REGION Network 17: Lift01 Y-Heber / Lift01 Y-Lift
   #sinstLift01_Y_Lift(iniHomePos := "FG_TS_Lift01_Y_Lift_InHome",   // "Cylinder_2Out2In"
                       iniWorkPos := "FG_TS_Lift01_Y_Lift_InWork",
                       actor := "TransportActors".Lift01_Lift,
                       signals := #signals,
                       manualMovement := #manualMovements,
                       homePos => "FG_TS_Lift01_Y_Lift_HomePos",
                       workPos => "FG_TS_Lift01_Y_Lift_WorkPos");
END_REGION

REGION Network 18: Lift01 M-Förderband / Lift01 M-Conveyor
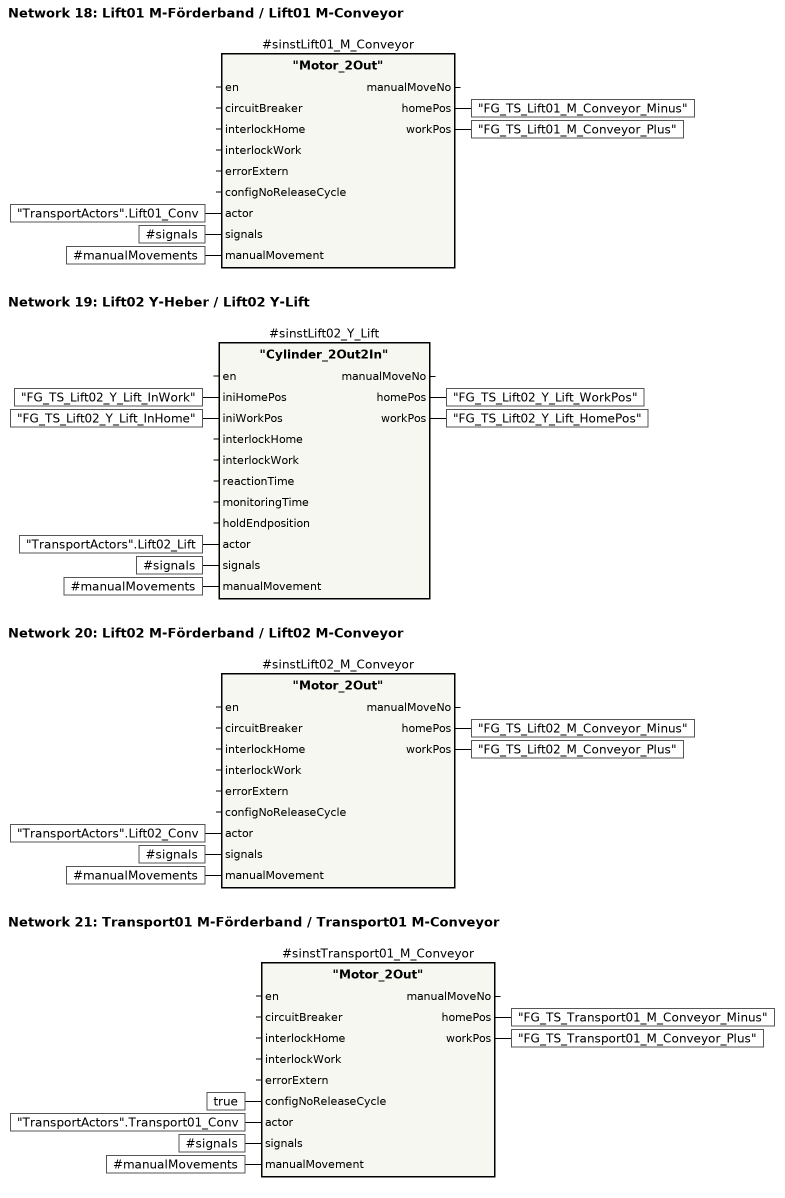
   #sinstLift01_M_Conveyor(actor := "TransportActors".Lift01_Conv,   // "Motor_2Out"
                           signals := #signals,
                           manualMovement := #manualMovements,
                           homePos => "FG_TS_Lift01_M_Conveyor_Minus",
                           workPos => "FG_TS_Lift01_M_Conveyor_Plus");
END_REGION

REGION Network 19: Lift02 Y-Heber / Lift02 Y-Lift
   #sinstLift02_Y_Lift(iniHomePos := "FG_TS_Lift02_Y_Lift_InWork",   // "Cylinder_2Out2In"
                       iniWorkPos := "FG_TS_Lift02_Y_Lift_InHome",
                       actor := "TransportActors".Lift02_Lift,
                       signals := #signals,
                       manualMovement := #manualMovements,
                       homePos => "FG_TS_Lift02_Y_Lift_WorkPos",
                       workPos => "FG_TS_Lift02_Y_Lift_HomePos");
END_REGION

REGION Network 20: Lift02 M-Förderband / Lift02 M-Conveyor
   #sinstLift02_M_Conveyor(actor := "TransportActors".Lift02_Conv,   // "Motor_2Out"
                           signals := #signals,
                           manualMovement := #manualMovements,
                           homePos => "FG_TS_Lift02_M_Conveyor_Minus",
                           workPos => "FG_TS_Lift02_M_Conveyor_Plus");
END_REGION

REGION Network 21: Transport01 M-Förderband / Transport01 M-Conveyor
   #sinstTransport01_M_Conveyor(configNoReleaseCycle := true,   // "Motor_2Out"
                           actor := "TransportActors".Transport01_Conv,
                           signals := #signals,
                           manualMovement := #manualMovements,
                           homePos => "FG_TS_Transport01_M_Conveyor_Minus",
                           workPos => "FG_TS_Transport01_M_Conveyor_Plus");
END_REGION

REGION Network 22: Transport02 M-Förderband / Transport02 M-Conveyor
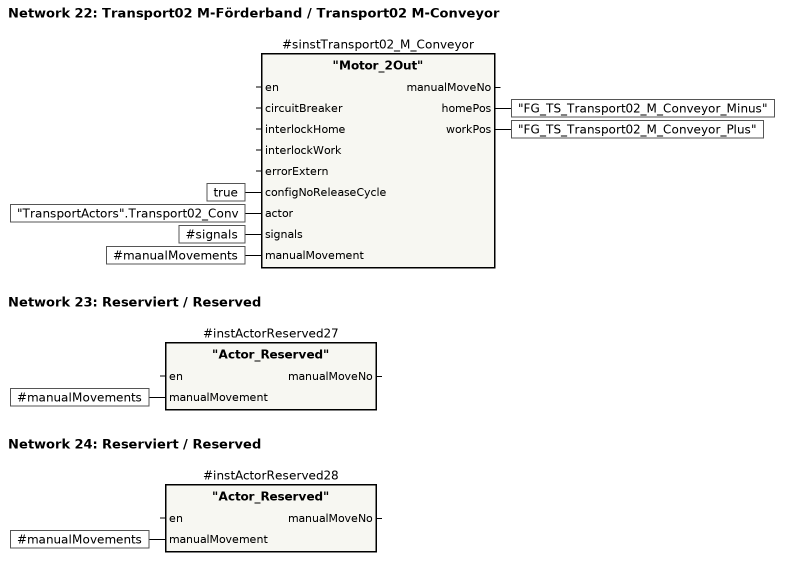
   #sinstTransport02_M_Conveyor(configNoReleaseCycle := true,   // "Motor_2Out"
                           actor := "TransportActors".Transport02_Conv,
                           signals := #signals,
                           manualMovement := #manualMovements,
                           homePos => "FG_TS_Transport02_M_Conveyor_Minus",
                           workPos => "FG_TS_Transport02_M_Conveyor_Plus");
END_REGION

REGION Network 23: Reserviert / Reserved
   #instActorReserved27(manualMovement := #manualMovements);   // "Actor_Reserved"
END_REGION

REGION Network 24: Reserviert / Reserved
   #instActorReserved28(manualMovement := #manualMovements);   // "Actor_Reserved"
END_REGION
END_FUNCTION_BLOCK

// folder: 2. Machine/10_FG_Transport/Stepsequences

FUNCTION "FG10StepSequences" : Void   // FC2010, FBD
TITLE = Schrittkettensteuerung / Sequence control
{ S7_Optimized_Access := 'TRUE' }
VERSION : 0.1
// Ersteller: Andreas Fast Automation
// Kontakt per LinkedIn: https://www.linkedin.com/in/automation-fast-andreas/
// 
// Das Projekt dient zu Demonstrationszwecken und kann frei genutzt werden.
// 
// Bausteinbeschreibung:
// Author: Andreas Fast Automation
// Kontakt per LinkedIn: https://www.linkedin.com/in/automation-fast-andreas/
// 
// This project is intended for demonstration purposes and may be used freely.
// 
// Block description:
   VAR_IN_OUT
      station : "typeStation";
   END_VAR
   VAR_TEMP
      tempInit : Bool;
      tempAck : Bool;
      tempSwAuto : Bool;
      tempSwMan : Bool;
      tempSwTap : Bool;
      tempPush : Bool;
   END_VAR
BEGIN

REGION Network 1: GRAPH-Parameter / GRAPH parameters
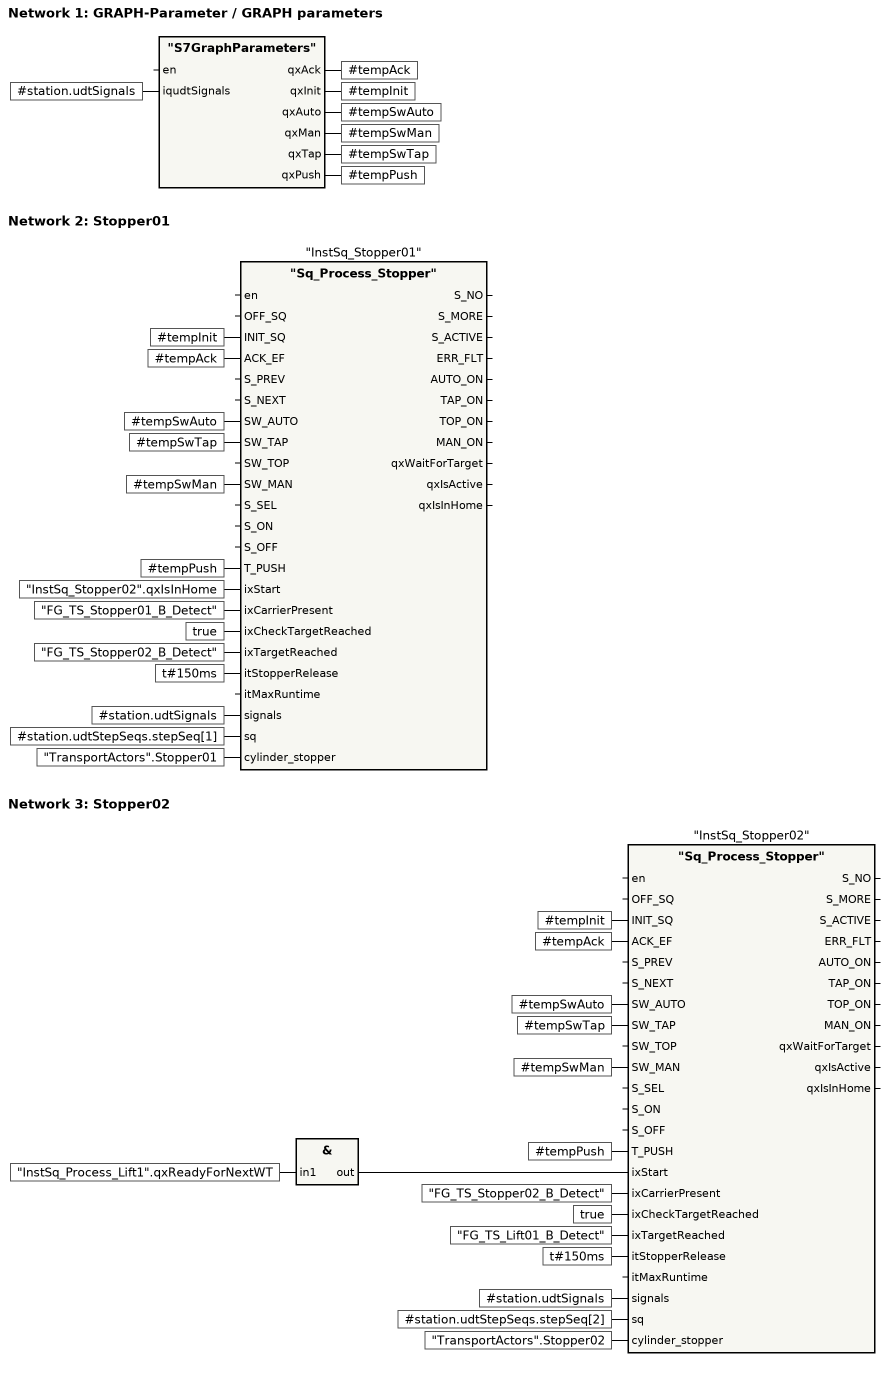
   "S7GraphParameters"(iqudtSignals := #station.udtSignals,
                       qxAck => #tempAck,
                       qxInit => #tempInit,
                       qxAuto => #tempSwAuto,
                       qxMan => #tempSwMan,
                       qxTap => #tempSwTap,
                       qxPush => #tempPush);
END_REGION

REGION Network 2: Stopper01
   "InstSq_Stopper01"(INIT_SQ := #tempInit,   // "Sq_Process_Stopper"
                      ACK_EF := #tempAck,
                      SW_AUTO := #tempSwAuto,
                      SW_TAP := #tempSwTap,
                      SW_MAN := #tempSwMan,
                      T_PUSH := #tempPush,
                      ixStart := "InstSq_Stopper02".qxIsInHome,
                      ixCarrierPresent := "FG_TS_Stopper01_B_Detect",
                      ixCheckTargetReached := true,
                      ixTargetReached := "FG_TS_Stopper02_B_Detect",
                      itStopperRelease := t#150ms,
                      signals := #station.udtSignals,
                      sq := #station.udtStepSeqs.stepSeq[1],
                      cylinder_stopper := "TransportActors".Stopper01);
END_REGION

REGION Network 3: Stopper02
   "InstSq_Stopper02"(INIT_SQ := #tempInit,   // "Sq_Process_Stopper"
                      ACK_EF := #tempAck,
                      SW_AUTO := #tempSwAuto,
                      SW_TAP := #tempSwTap,
                      SW_MAN := #tempSwMan,
                      T_PUSH := #tempPush,
                      ixStart := "InstSq_Process_Lift1".qxReadyForNextWT,
                      ixCarrierPresent := "FG_TS_Stopper02_B_Detect",
                      ixCheckTargetReached := true,
                      ixTargetReached := "FG_TS_Lift01_B_Detect",
                      itStopperRelease := t#150ms,
                      signals := #station.udtSignals,
                      sq := #station.udtStepSeqs.stepSeq[2],
                      cylinder_stopper := "TransportActors".Stopper02);
END_REGION

REGION Network 4: Lift 1
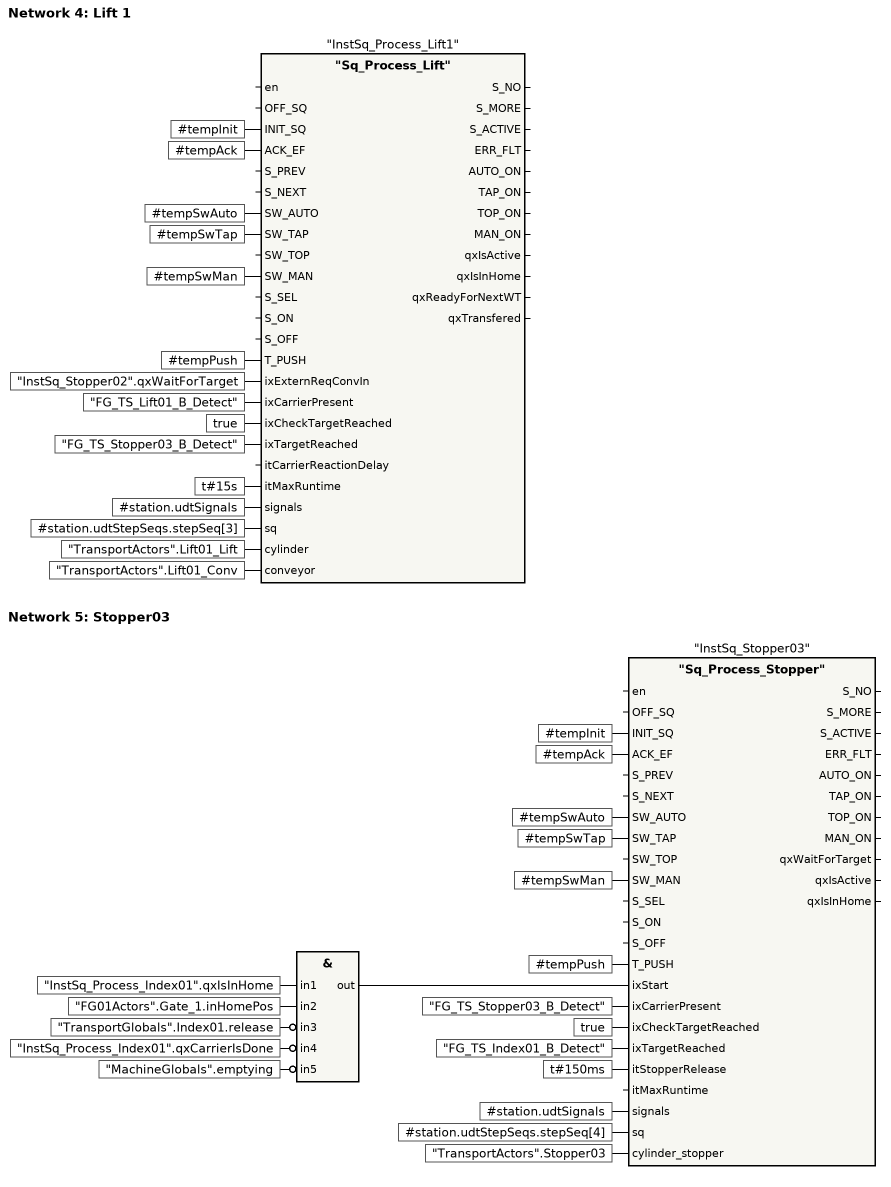
   "InstSq_Process_Lift1"(INIT_SQ := #tempInit,   // "Sq_Process_Lift"
                          ACK_EF := #tempAck,
                          SW_AUTO := #tempSwAuto,
                          SW_TAP := #tempSwTap,
                          SW_MAN := #tempSwMan,
                          T_PUSH := #tempPush,
                          ixExternReqConvIn := "InstSq_Stopper02".qxWaitForTarget,
                          ixCarrierPresent := "FG_TS_Lift01_B_Detect",
                          ixCheckTargetReached := true,
                          ixTargetReached := "FG_TS_Stopper03_B_Detect",
                          itMaxRuntime := t#15s,
                          signals := #station.udtSignals,
                          sq := #station.udtStepSeqs.stepSeq[3],
                          cylinder := "TransportActors".Lift01_Lift,
                          conveyor := "TransportActors".Lift01_Conv);
END_REGION

REGION Network 5: Stopper03
   "InstSq_Stopper03"(INIT_SQ := #tempInit,   // "Sq_Process_Stopper"
                      ACK_EF := #tempAck,
                      SW_AUTO := #tempSwAuto,
                      SW_TAP := #tempSwTap,
                      SW_MAN := #tempSwMan,
                      T_PUSH := #tempPush,
                      ixStart := "InstSq_Process_Index01".qxIsInHome AND "FG01Actors".Gate_1.inHomePos AND NOT "TransportGlobals".Index01.release AND NOT "InstSq_Process_Index01".qxCarrierIsDone AND NOT "MachineGlobals".emptying,
                      ixCarrierPresent := "FG_TS_Stopper03_B_Detect",
                      ixCheckTargetReached := true,
                      ixTargetReached := "FG_TS_Index01_B_Detect",
                      itStopperRelease := t#150ms,
                      signals := #station.udtSignals,
                      sq := #station.udtStepSeqs.stepSeq[4],
                      cylinder_stopper := "TransportActors".Stopper03);
END_REGION

REGION Network 6: Index01
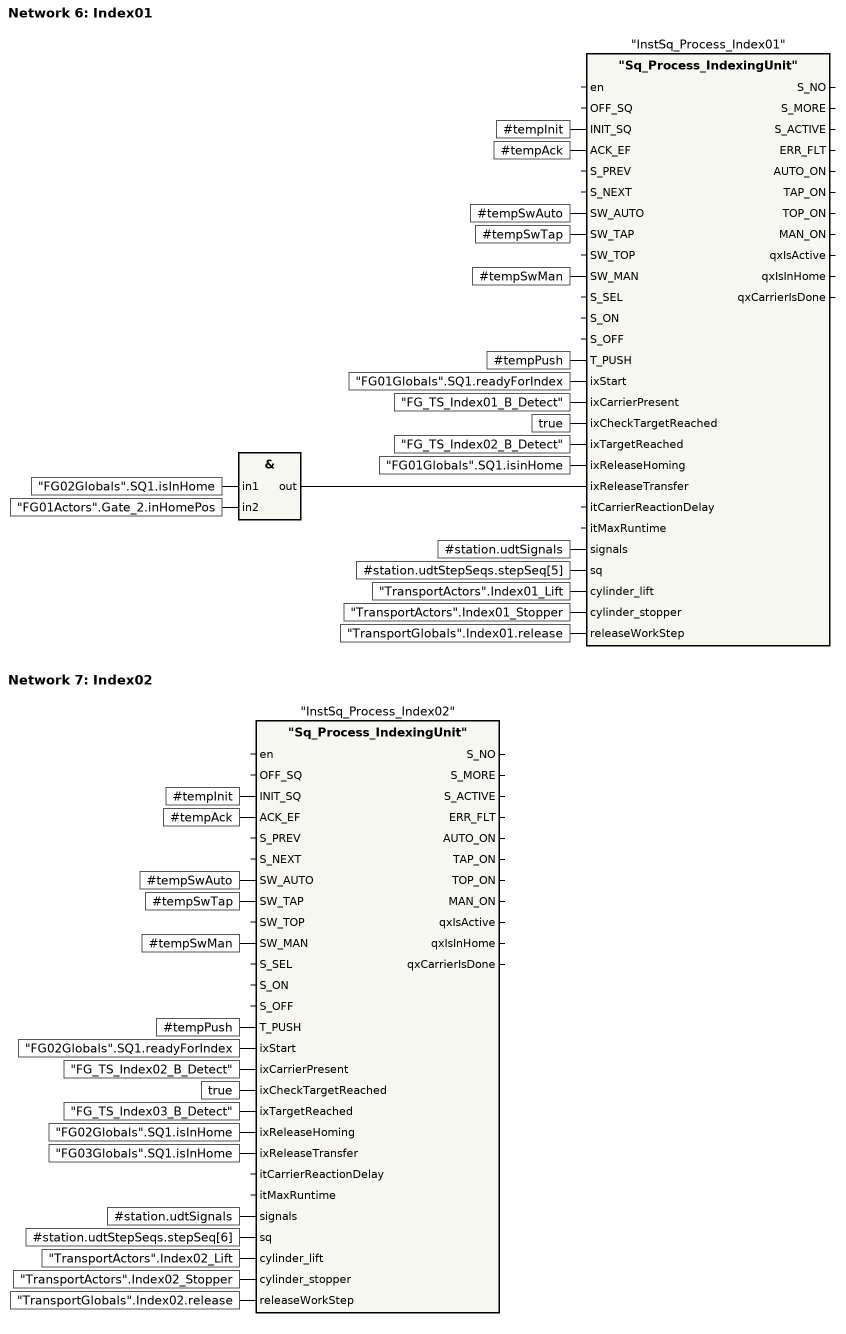
   "InstSq_Process_Index01"(INIT_SQ := #tempInit,   // "Sq_Process_IndexingUnit"
                           ACK_EF := #tempAck,
                           SW_AUTO := #tempSwAuto,
                           SW_TAP := #tempSwTap,
                           SW_MAN := #tempSwMan,
                           T_PUSH := #tempPush,
                           ixStart := "FG01Globals".SQ1.readyForIndex,
                           ixCarrierPresent := "FG_TS_Index01_B_Detect",
                           ixCheckTargetReached := true,
                           ixTargetReached := "FG_TS_Index02_B_Detect",
                           ixReleaseHoming := "FG01Globals".SQ1.isinHome,
                           ixReleaseTransfer := "FG02Globals".SQ1.isInHome AND "FG01Actors".Gate_2.inHomePos,
                           signals := #station.udtSignals,
                           sq := #station.udtStepSeqs.stepSeq[5],
                           cylinder_lift := "TransportActors".Index01_Lift,
                           cylinder_stopper := "TransportActors".Index01_Stopper,
                           releaseWorkStep := "TransportGlobals".Index01.release);
END_REGION

REGION Network 7: Index02
   "InstSq_Process_Index02"(INIT_SQ := #tempInit,   // "Sq_Process_IndexingUnit"
                           ACK_EF := #tempAck,
                           SW_AUTO := #tempSwAuto,
                           SW_TAP := #tempSwTap,
                           SW_MAN := #tempSwMan,
                           T_PUSH := #tempPush,
                           ixStart := "FG02Globals".SQ1.readyForIndex,
                           ixCarrierPresent := "FG_TS_Index02_B_Detect",
                           ixCheckTargetReached := true,
                           ixTargetReached := "FG_TS_Index03_B_Detect",
                           ixReleaseHoming := "FG02Globals".SQ1.isInHome,
                           ixReleaseTransfer := "FG03Globals".SQ1.isInHome,
                           signals := #station.udtSignals,
                           sq := #station.udtStepSeqs.stepSeq[6],
                           cylinder_lift := "TransportActors".Index02_Lift,
                           cylinder_stopper := "TransportActors".Index02_Stopper,
                           releaseWorkStep := "TransportGlobals".Index02.release);
END_REGION

REGION Network 8: Index03
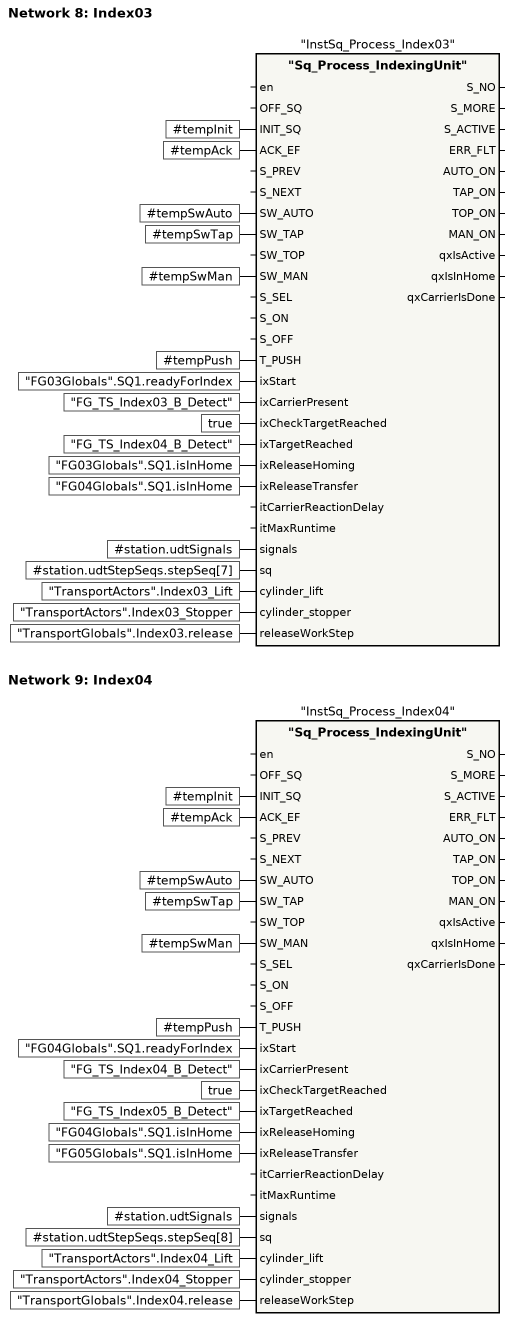
   "InstSq_Process_Index03"(INIT_SQ := #tempInit,   // "Sq_Process_IndexingUnit"
                           ACK_EF := #tempAck,
                           SW_AUTO := #tempSwAuto,
                           SW_TAP := #tempSwTap,
                           SW_MAN := #tempSwMan,
                           T_PUSH := #tempPush,
                           ixStart := "FG03Globals".SQ1.readyForIndex,
                           ixCarrierPresent := "FG_TS_Index03_B_Detect",
                           ixCheckTargetReached := true,
                           ixTargetReached := "FG_TS_Index04_B_Detect",
                           ixReleaseHoming := "FG03Globals".SQ1.isInHome,
                           ixReleaseTransfer := "FG04Globals".SQ1.isInHome,
                           signals := #station.udtSignals,
                           sq := #station.udtStepSeqs.stepSeq[7],
                           cylinder_lift := "TransportActors".Index03_Lift,
                           cylinder_stopper := "TransportActors".Index03_Stopper,
                           releaseWorkStep := "TransportGlobals".Index03.release);
END_REGION

REGION Network 9: Index04
   "InstSq_Process_Index04"(INIT_SQ := #tempInit,   // "Sq_Process_IndexingUnit"
                           ACK_EF := #tempAck,
                           SW_AUTO := #tempSwAuto,
                           SW_TAP := #tempSwTap,
                           SW_MAN := #tempSwMan,
                           T_PUSH := #tempPush,
                           ixStart := "FG04Globals".SQ1.readyForIndex,
                           ixCarrierPresent := "FG_TS_Index04_B_Detect",
                           ixCheckTargetReached := true,
                           ixTargetReached := "FG_TS_Index05_B_Detect",
                           ixReleaseHoming := "FG04Globals".SQ1.isInHome,
                           ixReleaseTransfer := "FG05Globals".SQ1.isInHome,
                           signals := #station.udtSignals,
                           sq := #station.udtStepSeqs.stepSeq[8],
                           cylinder_lift := "TransportActors".Index04_Lift,
                           cylinder_stopper := "TransportActors".Index04_Stopper,
                           releaseWorkStep := "TransportGlobals".Index04.release);
END_REGION

REGION Network 10: Index05
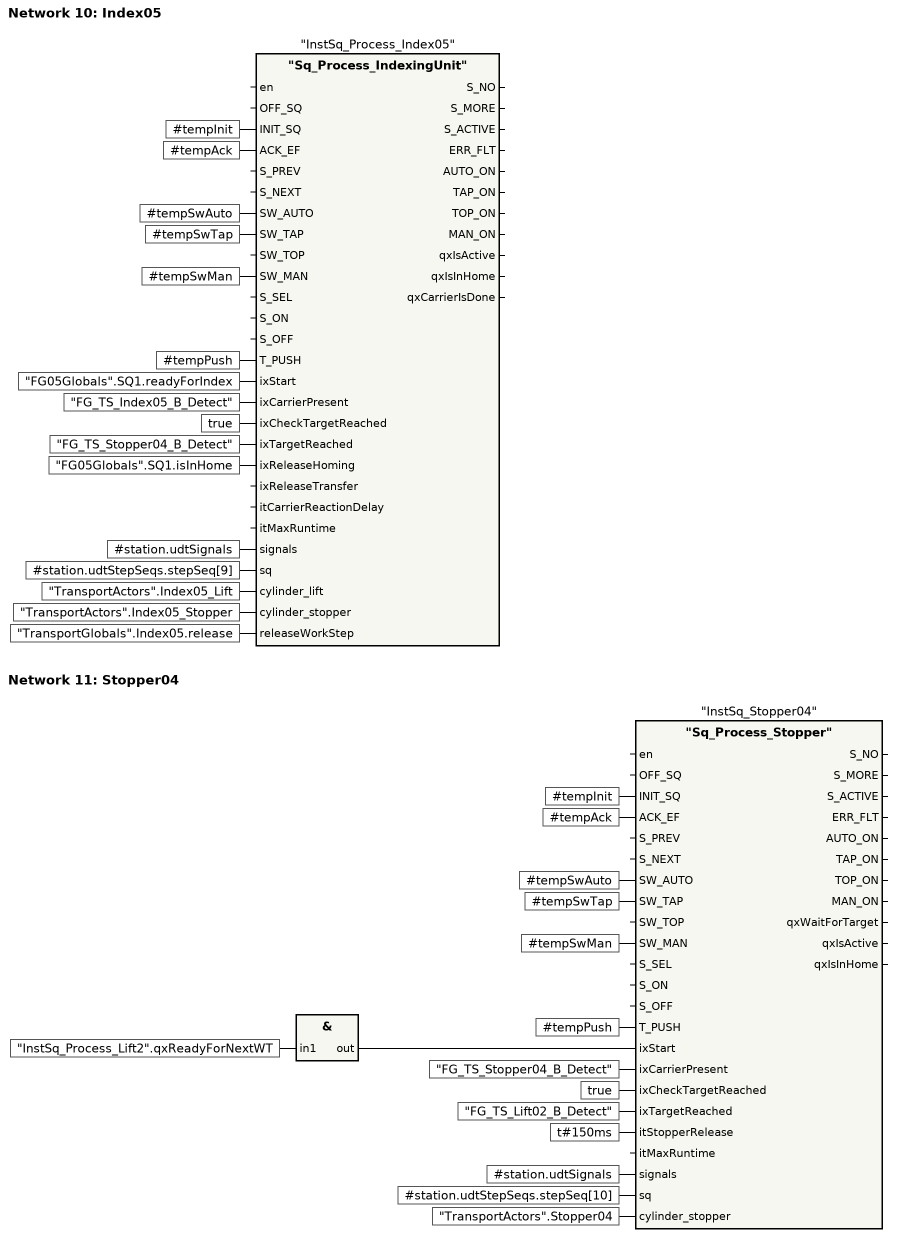
   "InstSq_Process_Index05"(INIT_SQ := #tempInit,   // "Sq_Process_IndexingUnit"
                           ACK_EF := #tempAck,
                           SW_AUTO := #tempSwAuto,
                           SW_TAP := #tempSwTap,
                           SW_MAN := #tempSwMan,
                           T_PUSH := #tempPush,
                           ixStart := "FG05Globals".SQ1.readyForIndex,
                           ixCarrierPresent := "FG_TS_Index05_B_Detect",
                           ixCheckTargetReached := true,
                           ixTargetReached := "FG_TS_Stopper04_B_Detect",
                           ixReleaseHoming := "FG05Globals".SQ1.isInHome,
                           signals := #station.udtSignals,
                           sq := #station.udtStepSeqs.stepSeq[9],
                           cylinder_lift := "TransportActors".Index05_Lift,
                           cylinder_stopper := "TransportActors".Index05_Stopper,
                           releaseWorkStep := "TransportGlobals".Index05.release);
END_REGION

REGION Network 11: Stopper04
   "InstSq_Stopper04"(INIT_SQ := #tempInit,   // "Sq_Process_Stopper"
                      ACK_EF := #tempAck,
                      SW_AUTO := #tempSwAuto,
                      SW_TAP := #tempSwTap,
                      SW_MAN := #tempSwMan,
                      T_PUSH := #tempPush,
                      ixStart := "InstSq_Process_Lift2".qxReadyForNextWT,
                      ixCarrierPresent := "FG_TS_Stopper04_B_Detect",
                      ixCheckTargetReached := true,
                      ixTargetReached := "FG_TS_Lift02_B_Detect",
                      itStopperRelease := t#150ms,
                      signals := #station.udtSignals,
                      sq := #station.udtStepSeqs.stepSeq[10],
                      cylinder_stopper := "TransportActors".Stopper04);
END_REGION

REGION Network 12: Lift 2
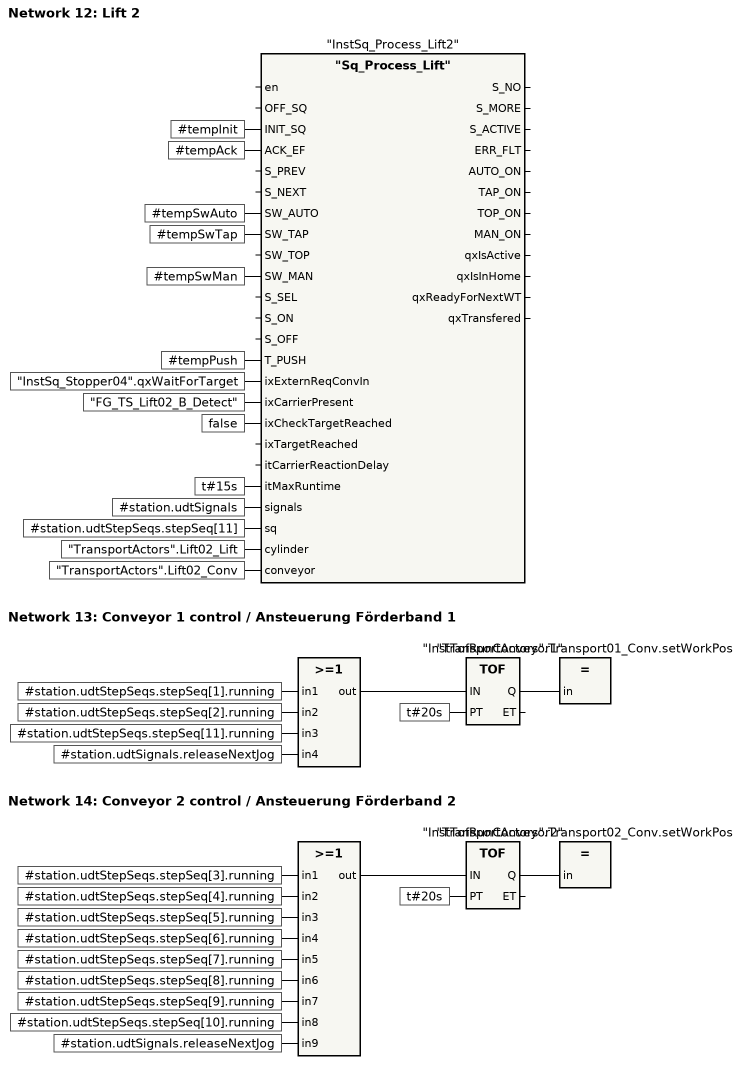
   "InstSq_Process_Lift2"(INIT_SQ := #tempInit,   // "Sq_Process_Lift"
                          ACK_EF := #tempAck,
                          SW_AUTO := #tempSwAuto,
                          SW_TAP := #tempSwTap,
                          SW_MAN := #tempSwMan,
                          T_PUSH := #tempPush,
                          ixExternReqConvIn := "InstSq_Stopper04".qxWaitForTarget,
                          ixCarrierPresent := "FG_TS_Lift02_B_Detect",
                          ixCheckTargetReached := false,
                          itMaxRuntime := t#15s,
                          signals := #station.udtSignals,
                          sq := #station.udtStepSeqs.stepSeq[11],
                          cylinder := "TransportActors".Lift02_Lift,
                          conveyor := "TransportActors".Lift02_Conv);
END_REGION

REGION Network 13: Conveyor 1 control / Ansteuerung Förderband 1
   "InstTofRunConveyor1".TOF(IN := #station.udtStepSeqs.stepSeq[1].running OR #station.udtStepSeqs.stepSeq[2].running OR #station.udtStepSeqs.stepSeq[11].running OR #station.udtSignals.releaseNextJog,
                           PT := t#20s);
   "TransportActors".Transport01_Conv.setWorkPos := "InstTofRunConveyor1".Q;
END_REGION

REGION Network 14: Conveyor 2 control / Ansteuerung Förderband 2
   "InstTofRunConveyor2".TOF(IN := #station.udtStepSeqs.stepSeq[3].running OR #station.udtStepSeqs.stepSeq[4].running OR #station.udtStepSeqs.stepSeq[5].running OR #station.udtStepSeqs.stepSeq[6].running OR #station.udtStepSeqs.stepSeq[7].running OR #station.udtStepSeqs.stepSeq[8].running OR #station.udtStepSeqs.stepSeq[9].running OR #station.udtStepSeqs.stepSeq[10].running OR #station.udtSignals.releaseNextJog,
                           PT := t#20s);
   "TransportActors".Transport02_Conv.setWorkPos := "InstTofRunConveyor2".Q;
END_REGION
END_FUNCTION

// folder: 9. Library/9.1 Framework Functions

FUNCTION "SetError" : Void   // FC900, FBD
TITLE = Setze Fehler / Set fault
{ S7_Optimized_Access := 'TRUE' }
VERSION : 0.1
// Ersteller: Andreas Fast Automation
// Kontakt per LinkedIn: https://www.linkedin.com/in/automation-fast-andreas/
// 
// Das Projekt dient zu Demonstrationszwecken und kann frei genutzt werden.
// 
// Bausteinbeschreibung:
// Author: Andreas Fast Automation
// Kontakt per LinkedIn: https://www.linkedin.com/in/automation-fast-andreas/
// 
// This project is intended for demonstration purposes and may be used freely.
// 
// Block description:
   VAR_INPUT
      ixTrigger : Bool;   // Auslöser / Trigger
      ixLogic : Bool;   // Auslöserlogik; 0 = trigger ausgelöst bei false / Trigger logic; 0 = Trigger activated when false
   END_VAR
   VAR_OUTPUT
      qxError : Bool;
   END_VAR
BEGIN

REGION Network 1
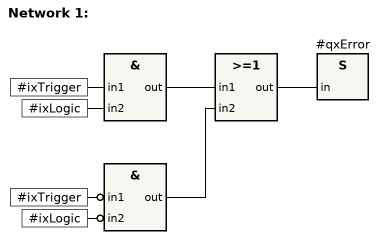
   IF (#ixTrigger AND #ixLogic) OR (NOT #ixTrigger AND NOT #ixLogic) THEN #qxError := TRUE; END_IF;
END_REGION
END_FUNCTION

FUNCTION "S7GraphParameters" : Void   // FC910, FBD
TITLE = Steuerung der GRAPH-Parameter / GRAPH parameter control
{ S7_Optimized_Access := 'TRUE' }
VERSION : 0.1
// Ersteller: Andreas Fast Automation
// Kontakt per LinkedIn: https://www.linkedin.com/in/automation-fast-andreas/
// 
// Das Projekt dient zu Demonstrationszwecken und kann frei genutzt werden.
// 
// Bausteinbeschreibung:
// Author: Andreas Fast Automation
// Kontakt per LinkedIn: https://www.linkedin.com/in/automation-fast-andreas/
// 
// This project is intended for demonstration purposes and may be used freely.
// 
// Block description:
   VAR_OUTPUT
      qxAck : Bool;   // Schrittkette quittieren / Acknowledge sequence
      qxInit : Bool;   // Schrittkette in Initialschritt schalten / Switch sequence to initial step
      qxAuto : Bool;   // Automatikbetrieb / Automatic operation
      qxMan : Bool;   // Handbetrieb / Manual operation
      qxTap : Bool;   // Halbautomatischer Betrieb / Semi-automatic operation
      qxPush : Bool;   // Schaltfreigabe für Transition im halbautomatischen Betrieb / Transition enable in semi-automatic operation
   END_VAR
   VAR_IN_OUT
      iqudtSignals : "typeStationSignals";
   END_VAR
BEGIN

REGION Network 1: Schrittkette in Initialschritt schalten / Switch sequence to initial step
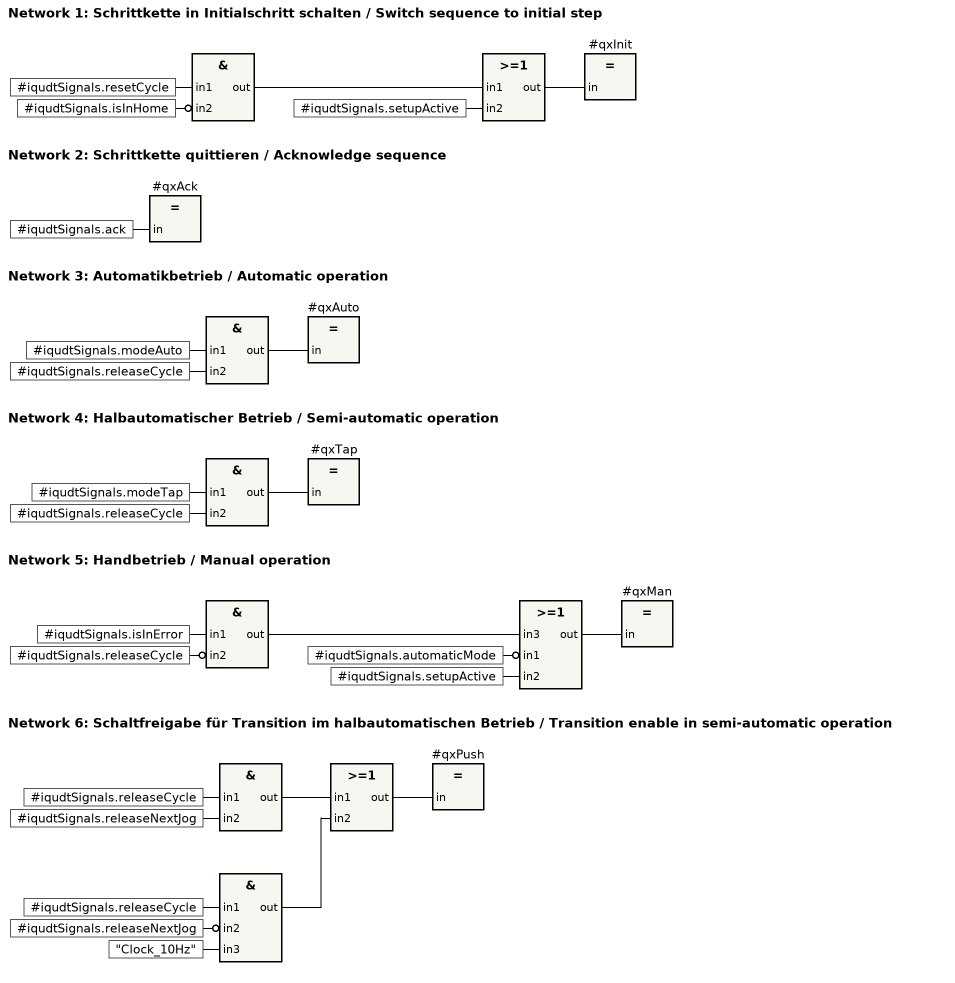
   #qxInit := (#iqudtSignals.resetCycle AND NOT #iqudtSignals.isInHome) OR #iqudtSignals.setupActive;
END_REGION

REGION Network 2: Schrittkette quittieren / Acknowledge sequence
   #qxAck := #iqudtSignals.ack;
END_REGION

REGION Network 3: Automatikbetrieb / Automatic operation
   #qxAuto := #iqudtSignals.modeAuto AND #iqudtSignals.releaseCycle;
END_REGION

REGION Network 4: Halbautomatischer Betrieb / Semi-automatic operation
   #qxTap := #iqudtSignals.modeTap AND #iqudtSignals.releaseCycle;
END_REGION

REGION Network 5: Handbetrieb / Manual operation
   #qxMan := (#iqudtSignals.isInError AND NOT #iqudtSignals.releaseCycle) OR NOT #iqudtSignals.automaticMode OR #iqudtSignals.setupActive;
END_REGION

REGION Network 6: Schaltfreigabe für Transition im halbautomatischen Betrieb / Transition enable in semi-automatic operation
   #qxPush := (#iqudtSignals.releaseCycle AND #iqudtSignals.releaseNextJog) OR (#iqudtSignals.releaseCycle AND NOT #iqudtSignals.releaseNextJog AND "Clock_10Hz");
END_REGION
END_FUNCTION

FUNCTION "S7GraphInterlock" : Void   // FC919, FBD
TITLE = S7G Verriegelung (notwendig für den Einzelschritt) / S7G interlock (required for single-step mode)
{ S7_Optimized_Access := 'TRUE' }
VERSION : 0.1
// Ersteller: Andreas Fast Automation
// Kontakt per LinkedIn: https://www.linkedin.com/in/automation-fast-andreas/
// 
// Das Projekt dient zu Demonstrationszwecken und kann frei genutzt werden.
// 
// Bausteinbeschreibung:
// Author: Andreas Fast Automation
// Kontakt per LinkedIn: https://www.linkedin.com/in/automation-fast-andreas/
// 
// This project is intended for demonstration purposes and may be used freely.
// 
// Block description:
   VAR_INPUT
      ixInterlock : Bool;   // Verriegelung / Interlock
      ixSetting : Bool;   // Verriegelungslogik (interlock == setting -> out wird freigegeben) / Interlock logic (interlock == setting -> out enabled)
      ixAlarm : Bool;   // Beim Alarm wird out rückgesetzt / out is reset on an alarm
   END_VAR
   VAR_OUTPUT
      qxOut : Bool;
   END_VAR
BEGIN

REGION Network 1
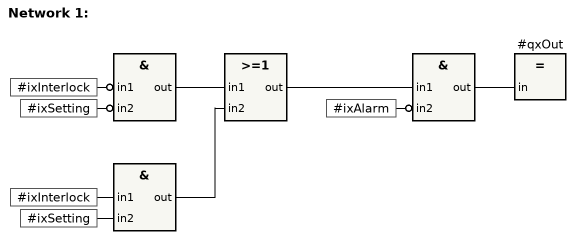
   #qxOut := ((NOT #ixInterlock AND NOT #ixSetting) OR (#ixInterlock AND #ixSetting)) AND NOT #ixAlarm;
END_REGION
END_FUNCTION

// folder: 9. Library/9.1 Framework Functions/01_Machine

FUNCTION_BLOCK "MachineControl"   // FB9000, FBD
TITLE = Maschinensteuerung / Machine control
{ S7_Optimized_Access := 'TRUE' }
VERSION : 0.1
// Ersteller: Andreas Fast Automation
// Kontakt per LinkedIn: https://www.linkedin.com/in/automation-fast-andreas/
// 
// Das Projekt dient zu Demonstrationszwecken und kann frei genutzt werden.
// 
// Bausteinbeschreibung:
// Author: Andreas Fast Automation
// Kontakt per LinkedIn: https://www.linkedin.com/in/automation-fast-andreas/
// 
// This project is intended for demonstration purposes and may be used freely.
// 
// Block description:
   VAR_INPUT
      ixFirstPlcCycle : Bool;   // Erster Zyklus / First cycle
      ixConfigNoControlOff : Bool := true;   // 1 = Ohne controlOff (Ein-/Ausschalten nur über controlOn) / 1 = Without controlOff (switch on/off using controlOn only)
      ixControlOn : Bool;   // Eingang „Steuerung ein“ (bei true) / Input 'control on' (if true)
      ixContolOff : Bool := true;   // Eingang „Steuerung aus“ (bei false) / Input 'control off' (if false)
      ixAutomaticMode : Bool;   // Eingang „Automatik-/Handbetrieb“ / Input 'automatic/manual operation'
      ixSingleStep : Bool;   // Eingang „Einzelschritt“ / Input 'single step'
      ixAutoStart : Bool;   // Eingang „Automatikstart“ / Input 'automatic start'
      ixAutoStop : Bool;   // Eingang „Automatikstopp“ / Input 'automatic stop'
      ixImmediateStop : Bool;   // Eingang „Sofort-Halt“ / Input 'immediate stop'
      ixReset : Bool;   // Eingang „Maschine zurücksetzen“ / Input 'machine reset'
      ixAcknowledge : Bool;   // Eingang „Quittierung“ / Input 'acknowledgement'
      ixErrFlt : Bool;   // Eingang „Maschinenstörung“ / Input 'machine fault'
      ixExternDevicesReady : Bool := true;   // Externe Geräte sind hochgefahren / External devices started up
   END_VAR
   VAR_OUTPUT
      qxControlOnLight : Bool;   // Steuerung Ein = Dauerlicht; Steuerung fährt hoch = Blinklicht; Steuerung aus = Licht aus / Control on = Steady light; control starting up = Flashing light; control off = Light off
      qxSetupOnLight : Bool;   // Einrichten aktiv = Ein / Setup active = On
      qxAutomaticRunsLight : Bool;   // Automatik aktiv = Dauerlicht; Teilautomatik = Blinklicht; Automatik aus = Licht aus / Automatic active = Steady light; semi-automatic = Flashing light; automatic off = Light off
      qxSingleStepLight : Bool;   // Einzelschritt läuft = Dauerlicht / Single step running = Steady light
      qxAutomaticStopsLight : Bool;   // Automatik stoppt = Blinklicht, Automatik hat Haltepunkt erreicht = Dauerlicht / Automatic stopping = Flashing light; automatic operation has reached the stop point = Steady light
      qxErrFltLight : Bool;   // Störung = Dauerlicht / Fault = Steady light
      qxHomingLight : Bool;   // Grundstellungsfahrt läuft = Blinklicht; Maschine in Grundstellung = Dauerlicht / Homing in progress = Flashing light; machine in home position = Steady light
      qxManAutoLight : Bool;   // Auto = Dauerlicht, Hand = Licht aus / Automatic = Steady light; manual = Light off
   END_VAR
   VAR_IN_OUT
      iqudtSafety : "typeMachineSafety";
      iqudtMachine : "typeMachine";
      iqudtStations : "typeStations";
      iqudtManualMovement : "typeManualMovements";
      iqudtPlcErrMsg : "typePlcErrMsg";
      iqudtHmiErrMsg : "typeHmiErrMsg";
   END_VAR
   VAR
      sxTrigControlOn : Bool;
      sxTrigReset : Bool;
      sxTrigSingleStep : Bool;
      sxTrigAutoStart : Bool;
      sxTrigHomingDone : Bool;
      sxTrigRunUp : Bool;
      sxTrigRunUpFlag : Bool;
      sxFirstCycle : Bool;
      sxStationsAllStopped : Bool;
      sxStationsAllRunning : Bool;
      sxAnyStationInAutoRun : Bool;
      sinstAlarmHandler : "AlarmHandler";
   END_VAR
   VAR_TEMP
      txStationError : Bool;
      txStationsInSetup : Bool;
      txAnyJogIsActive : Bool;
      txAnyStationIsHoming : Bool;
   END_VAR
   VAR_TEMP   // added for the SCL form of the ladder/FBD networks
      _w1 : Bool;
      _w2 : Bool;
   END_VAR
BEGIN

REGION Network 1: Meldungen auslösen / Trigger messages
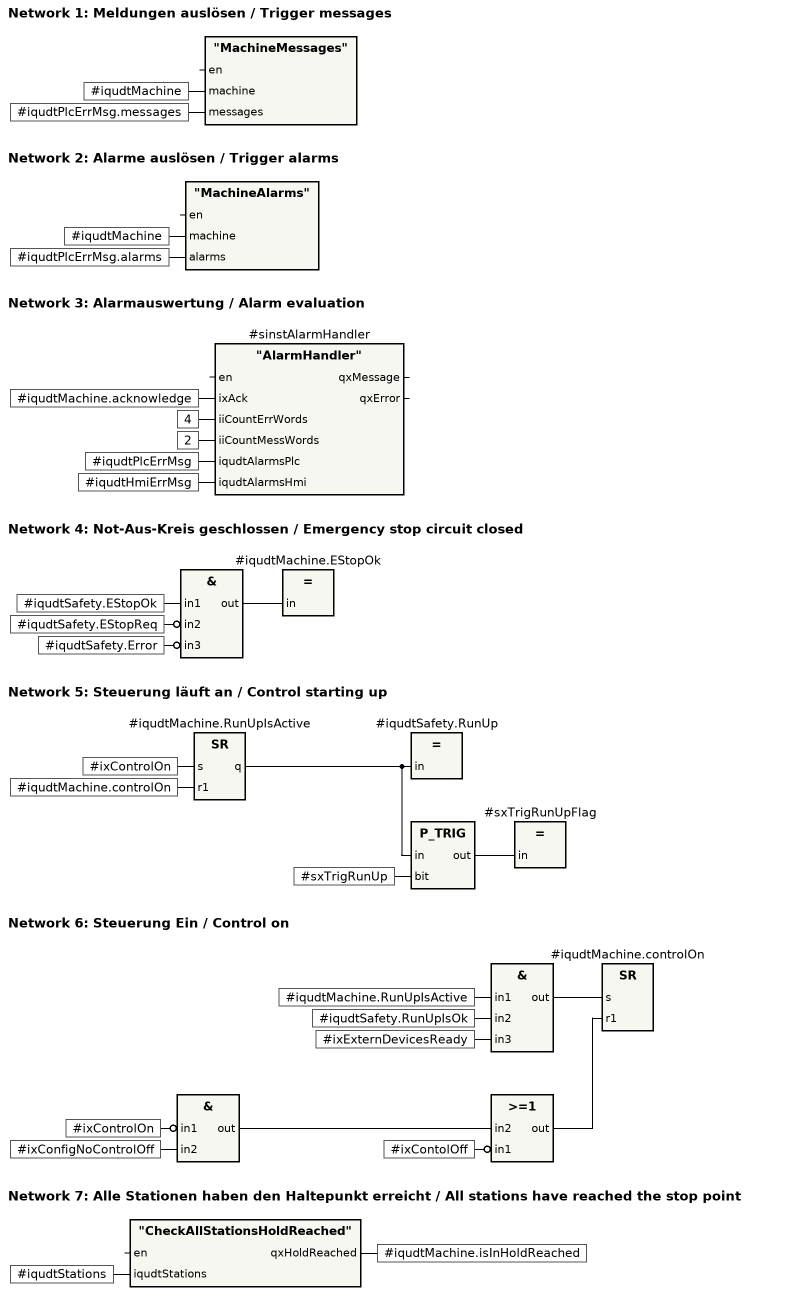
   "MachineMessages"(machine := #iqudtMachine, messages := #iqudtPlcErrMsg.messages);
END_REGION

REGION Network 2: Alarme auslösen / Trigger alarms
   "MachineAlarms"(machine := #iqudtMachine, alarms := #iqudtPlcErrMsg.alarms);
END_REGION

REGION Network 3: Alarmauswertung / Alarm evaluation
   #sinstAlarmHandler(ixAck := #iqudtMachine.acknowledge,   // "AlarmHandler"
                      iiCountErrWords := 4,
                      iiCountMessWords := 2,
                      iqudtAlarmsPlc := #iqudtPlcErrMsg,
                      iqudtAlarmsHmi := #iqudtHmiErrMsg);
END_REGION

REGION Network 4: Not-Aus-Kreis geschlossen / Emergency stop circuit closed
   #iqudtMachine.EStopOk := #iqudtSafety.EStopOk AND NOT #iqudtSafety.EStopReq AND NOT #iqudtSafety.Error;
END_REGION

REGION Network 5: Steuerung läuft an / Control starting up
   IF #ixControlOn THEN
       #iqudtMachine.RunUpIsActive := TRUE;   // SR flip-flop
   END_IF;
   IF #iqudtMachine.controlOn THEN #iqudtMachine.RunUpIsActive := FALSE; END_IF;
   #iqudtSafety.RunUp := #iqudtMachine.RunUpIsActive;
   #_w1 := #iqudtMachine.RunUpIsActive AND NOT #sxTrigRunUp;   // rising edge
   #sxTrigRunUp := #iqudtMachine.RunUpIsActive;
   #sxTrigRunUpFlag := #_w1;
END_REGION

REGION Network 6: Steuerung Ein / Control on
   IF #iqudtMachine.RunUpIsActive AND #iqudtSafety.RunUpIsOk AND #ixExternDevicesReady THEN
       #iqudtMachine.controlOn := TRUE;   // SR flip-flop
   END_IF;
   IF (NOT #ixControlOn AND #ixConfigNoControlOff) OR NOT #ixContolOff THEN
       #iqudtMachine.controlOn := FALSE;
   END_IF;
END_REGION

REGION Network 7: Alle Stationen haben den Haltepunkt erreicht / All stations have reached the stop point
   "CheckAllStationsHoldReached"(iqudtStations := #iqudtStations,
                           qxHoldReached => #iqudtMachine.isInHoldReached);
END_REGION

REGION Network 8: Alle Stationen stehen in Grundstellung / All stations in home position
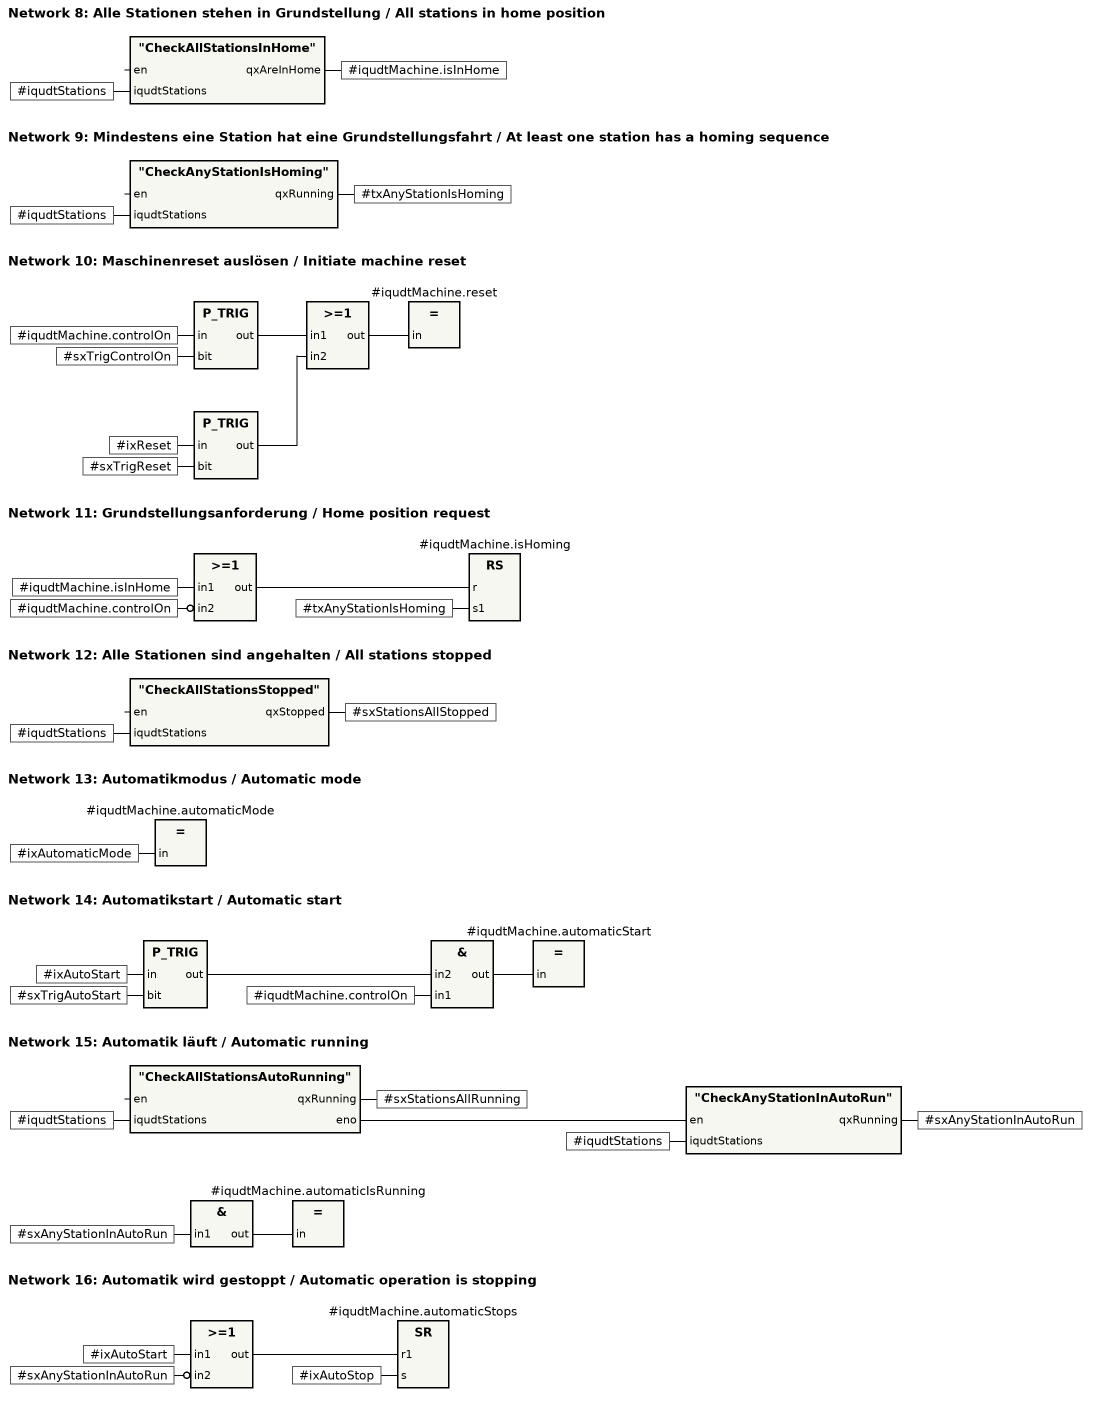
   "CheckAllStationsInHome"(iqudtStations := #iqudtStations, qxAreInHome => #iqudtMachine.isInHome);
END_REGION

REGION Network 9: Mindestens eine Station hat eine Grundstellungsfahrt / At least one station has a homing sequence
   "CheckAnyStationIsHoming"(iqudtStations := #iqudtStations, qxRunning => #txAnyStationIsHoming);
END_REGION

REGION Network 10: Maschinenreset auslösen / Initiate machine reset
   #_w1 := #iqudtMachine.controlOn AND NOT #sxTrigControlOn;   // rising edge
   #sxTrigControlOn := #iqudtMachine.controlOn;
   #_w2 := #ixReset AND NOT #sxTrigReset;   // rising edge
   #sxTrigReset := #ixReset;
   #iqudtMachine.reset := #_w1 OR #_w2;
END_REGION

REGION Network 11: Grundstellungsanforderung / Home position request
   IF #iqudtMachine.isInHome OR NOT #iqudtMachine.controlOn THEN
       #iqudtMachine.isHoming := FALSE;   // RS flip-flop
   END_IF;
   IF #txAnyStationIsHoming THEN #iqudtMachine.isHoming := TRUE; END_IF;
END_REGION

REGION Network 12: Alle Stationen sind angehalten / All stations stopped
   "CheckAllStationsStopped"(iqudtStations := #iqudtStations, qxStopped => #sxStationsAllStopped);
END_REGION

REGION Network 13: Automatikmodus / Automatic mode
   #iqudtMachine.automaticMode := #ixAutomaticMode;
END_REGION

REGION Network 14: Automatikstart / Automatic start
   #_w1 := #ixAutoStart AND NOT #sxTrigAutoStart;   // rising edge
   #sxTrigAutoStart := #ixAutoStart;
   #iqudtMachine.automaticStart := #_w1 AND #iqudtMachine.controlOn;
END_REGION

REGION Network 15: Automatik läuft / Automatic running
   "CheckAllStationsAutoRunning"(iqudtStations := #iqudtStations,
                           qxRunning => #sxStationsAllRunning,
                           ENO => #_w1);
   IF #_w1 THEN
       "CheckAnyStationInAutoRun"(iqudtStations := #iqudtStations, qxRunning => #sxAnyStationInAutoRun);
   END_IF;
   #iqudtMachine.automaticIsRunning := #sxAnyStationInAutoRun;
END_REGION

REGION Network 16: Automatik wird gestoppt / Automatic operation is stopping
   IF #ixAutoStop THEN
       #iqudtMachine.automaticStops := TRUE;   // SR flip-flop
   END_IF;
   IF #ixAutoStart OR NOT #sxAnyStationInAutoRun THEN #iqudtMachine.automaticStops := FALSE; END_IF;
END_REGION

REGION Network 17: Sofort Halt auslösen / Initiate immediate stop
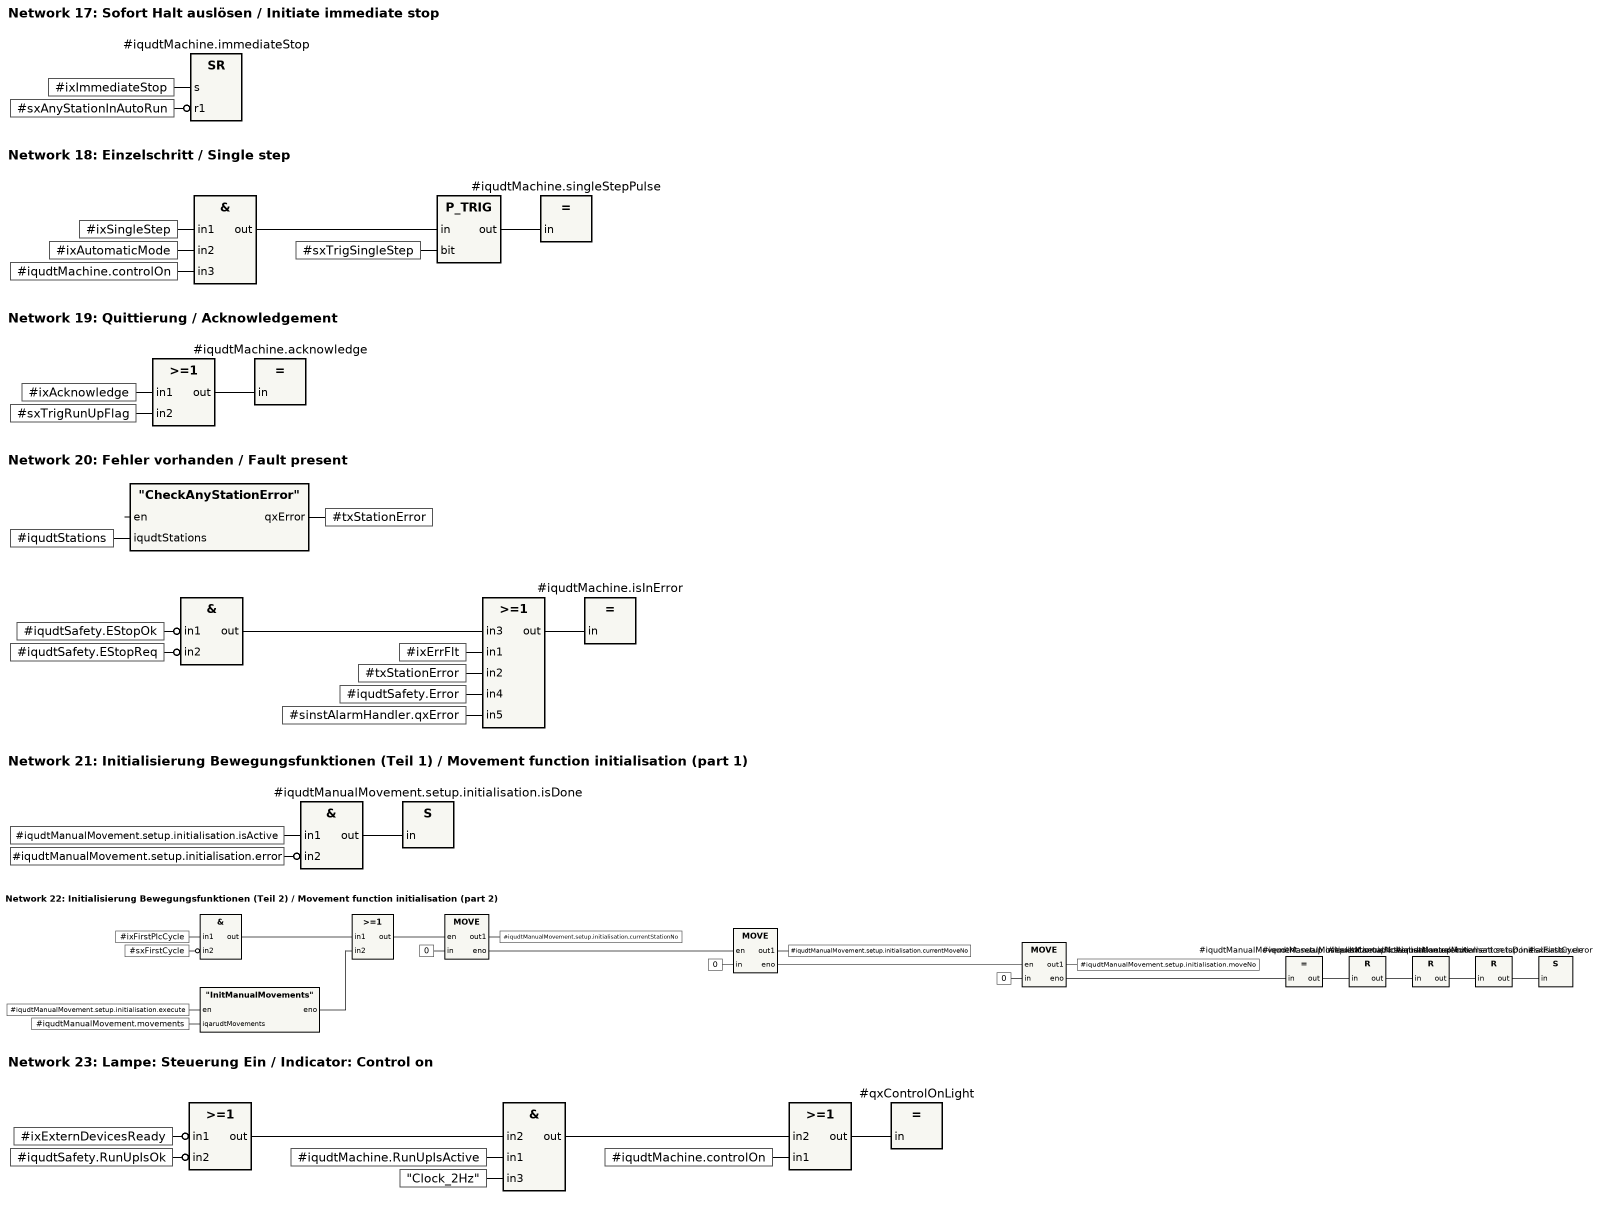
   IF #ixImmediateStop THEN
       #iqudtMachine.immediateStop := TRUE;   // SR flip-flop
   END_IF;
   IF NOT #sxAnyStationInAutoRun THEN #iqudtMachine.immediateStop := FALSE; END_IF;
END_REGION

REGION Network 18: Einzelschritt / Single step
   #_w1 := #ixSingleStep AND #ixAutomaticMode AND #iqudtMachine.controlOn;
   #_w2 := #_w1 AND NOT #sxTrigSingleStep;   // rising edge
   #sxTrigSingleStep := #_w1;
   #iqudtMachine.singleStepPulse := #_w2;
END_REGION

REGION Network 19: Quittierung / Acknowledgement
   #iqudtMachine.acknowledge := #ixAcknowledge OR #sxTrigRunUpFlag;
END_REGION

REGION Network 20: Fehler vorhanden / Fault present
   "CheckAnyStationError"(iqudtStations := #iqudtStations, qxError => #txStationError);
   #iqudtMachine.isInError := (NOT #iqudtSafety.EStopOk AND NOT #iqudtSafety.EStopReq) OR #ixErrFlt OR #txStationError OR #iqudtSafety.Error OR #sinstAlarmHandler.qxError;
END_REGION

REGION Network 21: Initialisierung Bewegungsfunktionen (Teil 1) / Movement function initialisation (part 1)
   IF #iqudtManualMovement.setup.initialisation.isActive AND NOT #iqudtManualMovement.setup.initialisation.error THEN
       #iqudtManualMovement.setup.initialisation.isDone := TRUE;
   END_IF;
END_REGION

REGION Network 22: Initialisierung Bewegungsfunktionen (Teil 2) / Movement function initialisation (part 2)
   "InitManualMovements"(EN := #iqudtManualMovement.setup.initialisation.execute,
                         iqarudtMovements := #iqudtManualMovement.movements,
                         ENO => #_w1);
   #_w2 := (#ixFirstPlcCycle AND NOT #sxFirstCycle) OR #_w1;
   IF #_w2 THEN
       #iqudtManualMovement.setup.initialisation.currentStationNo := 0;
       #iqudtManualMovement.setup.initialisation.currentMoveNo := 0;
       #iqudtManualMovement.setup.initialisation.moveNo := 0;
   END_IF;
   #iqudtManualMovement.setup.initialisation.isActive := #_w2;
   IF #_w2 THEN
       #iqudtManualMovement.setup.initialisation.execute := FALSE;
       #iqudtManualMovement.setup.initialisation.isDone := FALSE;
       #iqudtManualMovement.setup.initialisation.error := FALSE;
       #sxFirstCycle := TRUE;
   END_IF;
END_REGION

REGION Network 23: Lampe: Steuerung Ein / Indicator: Control on
   #qxControlOnLight := ((NOT #ixExternDevicesReady OR NOT #iqudtSafety.RunUpIsOk) AND #iqudtMachine.RunUpIsActive AND "Clock_2Hz") OR #iqudtMachine.controlOn;
END_REGION

REGION Network 24: Lampe: Einrichten aktiv / Indicator: Setup active
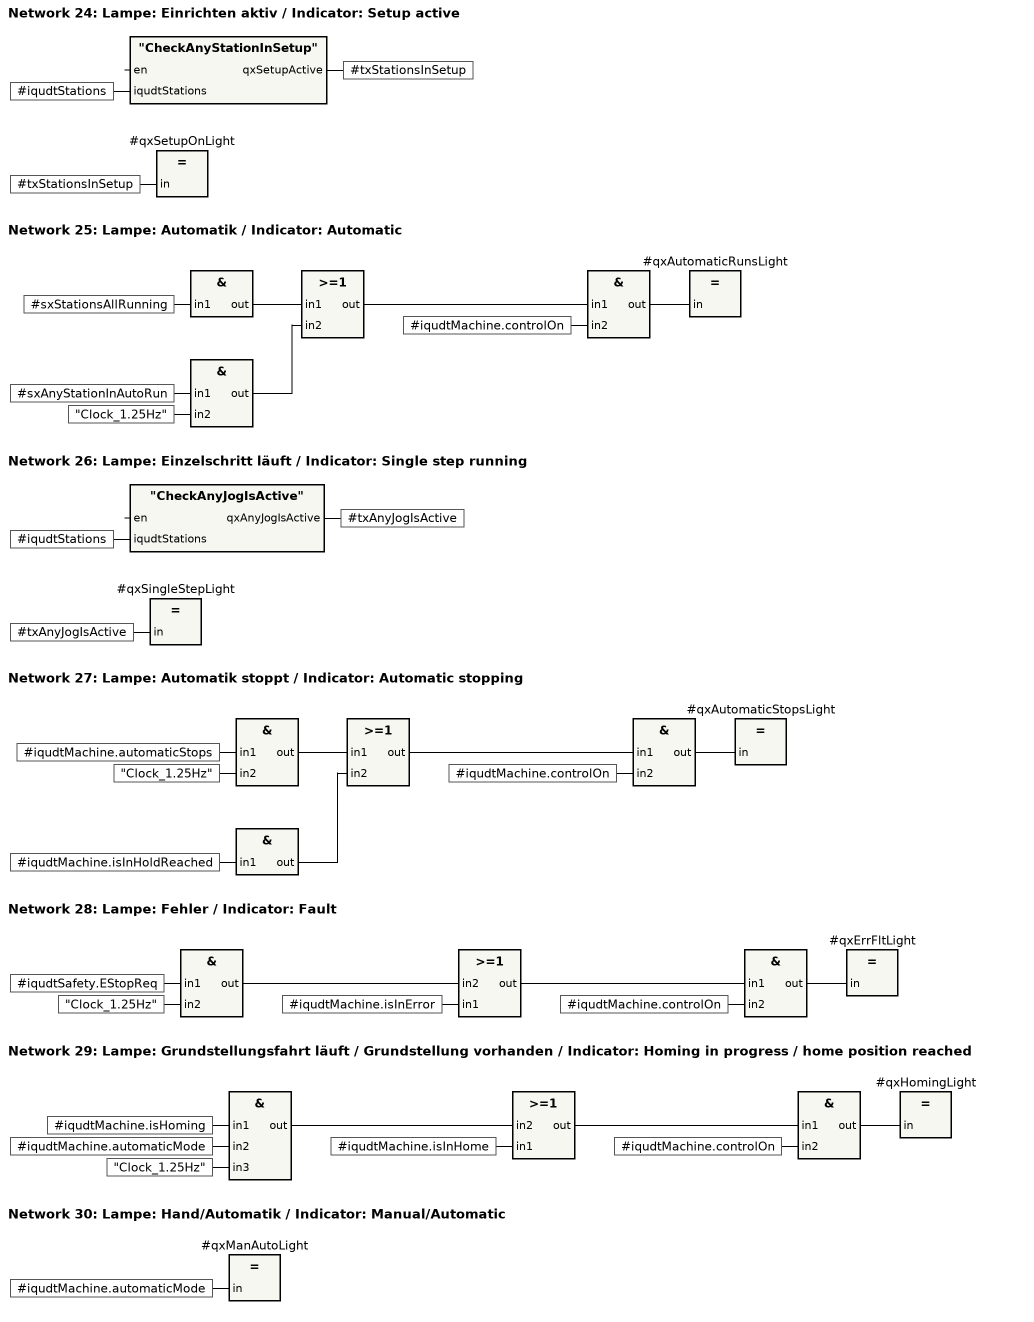
   "CheckAnyStationInSetup"(iqudtStations := #iqudtStations, qxSetupActive => #txStationsInSetup);
   #qxSetupOnLight := #txStationsInSetup;
END_REGION

REGION Network 25: Lampe: Automatik / Indicator: Automatic
   #qxAutomaticRunsLight := (#sxStationsAllRunning OR (#sxAnyStationInAutoRun AND "Clock_1.25Hz")) AND #iqudtMachine.controlOn;
END_REGION

REGION Network 26: Lampe: Einzelschritt läuft / Indicator: Single step running
   "CheckAnyJogIsActive"(iqudtStations := #iqudtStations, qxAnyJogIsActive => #txAnyJogIsActive);
   #qxSingleStepLight := #txAnyJogIsActive;
END_REGION

REGION Network 27: Lampe: Automatik stoppt / Indicator: Automatic stopping
   #qxAutomaticStopsLight := ((#iqudtMachine.automaticStops AND "Clock_1.25Hz") OR #iqudtMachine.isInHoldReached) AND #iqudtMachine.controlOn;
END_REGION

REGION Network 28: Lampe: Fehler / Indicator: Fault
   #qxErrFltLight := ((#iqudtSafety.EStopReq AND "Clock_1.25Hz") OR #iqudtMachine.isInError) AND #iqudtMachine.controlOn;
END_REGION

REGION Network 29: Lampe: Grundstellungsfahrt läuft / Grundstellung vorhanden / Indicator: Homing in progress / home position reached
   #qxHomingLight := ((#iqudtMachine.isHoming AND #iqudtMachine.automaticMode AND "Clock_1.25Hz") OR #iqudtMachine.isInHome) AND #iqudtMachine.controlOn;
END_REGION

REGION Network 30: Lampe: Hand/Automatik / Indicator: Manual/Automatic
   #qxManAutoLight := #iqudtMachine.automaticMode;
END_REGION
END_FUNCTION_BLOCK

FUNCTION "CheckAllStationsStopped" : Void   // FC901, SCL
{ S7_Optimized_Access := 'TRUE' }
VERSION : 0.1
   VAR_OUTPUT
      qxStopped : Bool;   // Alle Stationen sind angehalten / All stations stopped
   END_VAR
   VAR_IN_OUT
      iqudtStations : "typeStations";
   END_VAR
   VAR_TEMP
      tusiCounter : USInt;
   END_VAR
BEGIN
   // Ersteller: Andreas Fast Automation
   // Kontakt per LinkedIn: https://www.linkedin.com/in/automation-fast-andreas/
   //
   // Projekt dient zu Demonstrationszwecken und frei genutzt werden.
   //
   // Bausteinbeschreibung:
   // 

   #qxStopped := true;

   FOR #tusiCounter := 1 TO "SYS_MACHINE_MAXSTATIONS" DO
       // Check if all stations are stopped
       IF NOT #iqudtStations.station[#tusiCounter].udtSignals.isStopped AND #iqudtStations.station[#tusiCounter].xExists THEN
           #qxStopped := false;
           RETURN;
       END_IF;
   END_FOR;
END_FUNCTION

FUNCTION "CheckAnyStationError" : Void   // FC902, SCL
{ S7_Optimized_Access := 'TRUE' }
VERSION : 0.1
// Prüfen, ob eine Station eine Störung hat / Check whether any station has a fault
   VAR_OUTPUT
      qxError : Bool;
   END_VAR
   VAR_IN_OUT
      iqudtStations : "typeStations";
   END_VAR
   VAR_TEMP
      tusiCounter : USInt;
   END_VAR
BEGIN
   // Ersteller: Andreas Fast Automation
   // Kontakt per LinkedIn: https://www.linkedin.com/in/automation-fast-andreas/
   //
   // Projekt dient zu Demonstrationszwecken und frei genutzt werden.
   //
   // Bausteinbeschreibung:
   // 

   #qxError := false;

   FOR #tusiCounter := 1 TO "SYS_MACHINE_MAXSTATIONS" DO
       // Check for error in stations
       IF #iqudtStations.station[#tusiCounter].udtSignals.isInError AND #iqudtStations.station[#tusiCounter].xExists THEN
           #qxError := true;
           RETURN;
       END_IF;
   END_FOR;
END_FUNCTION

FUNCTION "CheckAnyStationInSetup" : Void   // FC903, SCL
{ S7_Optimized_Access := 'TRUE' }
VERSION : 0.1
// Prüfen, ob eine Station eine Störung hat / Check whether any station has a fault
   VAR_OUTPUT
      qxSetupActive : Bool;
   END_VAR
   VAR_IN_OUT
      iqudtStations : "typeStations";
   END_VAR
   VAR_TEMP
      tusiCounter : USInt;
   END_VAR
BEGIN
   // Ersteller: Andreas Fast Automation
   // Kontakt per LinkedIn: https://www.linkedin.com/in/automation-fast-andreas/
   //
   // Projekt dient zu Demonstrationszwecken und frei genutzt werden.
   //
   // Bausteinbeschreibung:
   // 

   #qxSetupActive := false;

   FOR #tusiCounter := 1 TO "SYS_MACHINE_MAXSTATIONS" DO
       // Check for error in stations
       IF #iqudtStations.station[#tusiCounter].udtSignals.setupActive AND #iqudtStations.station[#tusiCounter].xExists THEN
           #qxSetupActive := true;
           RETURN;
       END_IF;
   END_FOR;
END_FUNCTION

FUNCTION "CheckAllStationsInHome" : Void   // FC904, SCL
{ S7_Optimized_Access := 'TRUE' }
VERSION : 0.1
   VAR_OUTPUT
      qxAreInHome : Bool;   // Alle Stationen stehen in Grundstellung / All stations in home position
   END_VAR
   VAR_IN_OUT
      iqudtStations : "typeStations";
   END_VAR
   VAR_TEMP
      tusiCounter : USInt;
   END_VAR
BEGIN
   // Ersteller: Andreas Fast Automation
   // Kontakt per LinkedIn: https://www.linkedin.com/in/automation-fast-andreas/
   //
   // Projekt dient zu Demonstrationszwecken und frei genutzt werden.
   //
   // Bausteinbeschreibung:
   // 

   #qxAreInHome := true;

   FOR #tusiCounter := 1 TO "SYS_MACHINE_MAXSTATIONS" DO
       // Check if all stations are stopped
       IF NOT #iqudtStations.station[#tusiCounter].udtSignals.isInHome AND #iqudtStations.station[#tusiCounter].xExists THEN
           #qxAreInHome := false;
           RETURN ;
       END_IF;
   END_FOR;
END_FUNCTION

FUNCTION "CheckAllStationsAutoRunning" : Void   // FC905, SCL
{ S7_Optimized_Access := 'TRUE' }
VERSION : 0.1
   VAR_OUTPUT
      qxRunning : Bool;   // Alle Stationen im Automatikbetrieb / All stations in automatic operation
   END_VAR
   VAR_IN_OUT
      iqudtStations : "typeStations";
   END_VAR
   VAR_TEMP
      tusiCounter : USInt;
   END_VAR
BEGIN
   // Ersteller: Andreas Fast Automation
   // Kontakt per LinkedIn: https://www.linkedin.com/in/automation-fast-andreas/
   //
   // Projekt dient zu Demonstrationszwecken und frei genutzt werden.
   //
   // Bausteinbeschreibung:
   // 

   #qxRunning := true;

   FOR #tusiCounter := 1 TO "SYS_MACHINE_MAXSTATIONS" DO
       // Check if all stations are stopped
       IF NOT #iqudtStations.station[#tusiCounter].udtSignals.releaseCycle
           AND #iqudtStations.station[#tusiCounter].xExists
       THEN
           #qxRunning := false;
           RETURN;
       END_IF;
   END_FOR;
END_FUNCTION

FUNCTION "CheckAnyStationInAutoRun" : Void   // FC906, SCL
{ S7_Optimized_Access := 'TRUE' }
VERSION : 0.1
   VAR_OUTPUT
      qxRunning : Bool;   // Alle Stationen im Automatikbetrieb / All stations in automatic operation
   END_VAR
   VAR_IN_OUT
      iqudtStations : "typeStations";
   END_VAR
   VAR_TEMP
      tusiCounter : USInt;
   END_VAR
BEGIN
   // Ersteller: Andreas Fast Automation
   // Kontakt per LinkedIn: https://www.linkedin.com/in/automation-fast-andreas/
   //
   // Projekt dient zu Demonstrationszwecken und frei genutzt werden.
   //
   // Bausteinbeschreibung:
   // 

   #qxRunning := false;

   FOR #tusiCounter := 1 TO "SYS_MACHINE_MAXSTATIONS" DO
       // Check if all stations are stopped
       IF //#stations.station[#tempCounter].signals.modeAuto AND
           #iqudtStations.station[#tusiCounter].udtSignals.releaseCycle
           AND #iqudtStations.station[#tusiCounter].xExists
       THEN
           #qxRunning := true;
           RETURN;
       END_IF;
   END_FOR;
END_FUNCTION

FUNCTION "CheckAnyStationIsHoming" : Void   // FC908, SCL
{ S7_Optimized_Access := 'TRUE' }
VERSION : 0.1
   VAR_OUTPUT
      qxRunning : Bool;   // Alle Stationen im Automatikbetrieb / All stations in automatic operation
   END_VAR
   VAR_IN_OUT
      iqudtStations : "typeStations";
   END_VAR
   VAR_TEMP
      tusiCounter : USInt;
   END_VAR
BEGIN
   // Ersteller: Andreas Fast Automation
   // Kontakt per LinkedIn: https://www.linkedin.com/in/automation-fast-andreas/
   //
   // Projekt dient zu Demonstrationszwecken und frei genutzt werden.
   //
   // Bausteinbeschreibung:
   // 

   #qxRunning := false;

   FOR #tusiCounter := 1 TO "SYS_MACHINE_MAXSTATIONS" DO
       // Check if all stations are stopped
       IF #iqudtStations.station[#tusiCounter].udtSignals.isHoming
           AND #iqudtStations.station[#tusiCounter].xExists
       THEN
           #qxRunning := true;
           RETURN;
       END_IF;
   END_FOR;
END_FUNCTION

FUNCTION "CheckAnyJogIsActive" : Void   // FC915, SCL
{ S7_Optimized_Access := 'TRUE' }
VERSION : 0.1
   VAR_OUTPUT
      qxAnyJogIsActive : Bool;   // Mindestens eine Schrittkette läuft noch in halbautomatischer Weiterschaltung / At least one sequence still executing semi-automatic step advance
   END_VAR
   VAR_IN_OUT
      iqudtStations : "typeStations";
   END_VAR
   VAR_TEMP
      tusiCounter : USInt;
   END_VAR
BEGIN
   // Ersteller: Andreas Fast Automation
   // Kontakt per LinkedIn: https://www.linkedin.com/in/automation-fast-andreas/
   //
   // Projekt dient zu Demonstrationszwecken und frei genutzt werden.
   //
   // Bausteinbeschreibung:
   // 

   #qxAnyJogIsActive := false;

   FOR #tusiCounter := 1 TO "SYS_MACHINE_MAXSTATIONS" DO

       IF #iqudtStations.station[#tusiCounter].xExists AND
           #iqudtStations.station[#tusiCounter].udtSignals.modeTap AND
           #iqudtStations.station[#tusiCounter].udtSignals.releaseCycle
       THEN
           #qxAnyJogIsActive := true;
           RETURN;
       END_IF;

   END_FOR;
END_FUNCTION

FUNCTION "CheckAllStationsHoldReached" : Void   // FC916, SCL
{ S7_Optimized_Access := 'TRUE' }
VERSION : 0.1
   VAR_OUTPUT
      qxHoldReached : Bool;   // Alle Stationen haben den Haltepunkt erreicht / All stations have reached the stop point
   END_VAR
   VAR_IN_OUT
      iqudtStations : "typeStations";
   END_VAR
   VAR_TEMP
      tusiCounter : USInt;
   END_VAR
BEGIN
   // Ersteller: Andreas Fast Automation
   // Kontakt per LinkedIn: https://www.linkedin.com/in/automation-fast-andreas/
   //
   // Projekt dient zu Demonstrationszwecken und frei genutzt werden.
   //
   // Bausteinbeschreibung:
   // 

   #qxHoldReached := true;

   FOR #tusiCounter := 1 TO "SYS_MACHINE_MAXSTATIONS" DO
       // Check if all stations are stopped
       IF NOT #iqudtStations.station[#tusiCounter].udtSignals.isInHoldReached AND #iqudtStations.station[#tusiCounter].xExists THEN
           #qxHoldReached := false;
           RETURN;
       END_IF;
   END_FOR;
END_FUNCTION

// folder: 9. Library/9.1 Framework Functions/02_Station

FUNCTION_BLOCK "StationControl"   // FB9001, FBD
TITLE = Steuerung Station / Station control
{ S7_Optimized_Access := 'TRUE' }
VERSION : 0.1
// Ersteller: Andreas Fast Automation
// Kontakt per LinkedIn: https://www.linkedin.com/in/automation-fast-andreas/
// 
// Das Projekt dient zu Demonstrationszwecken und kann frei genutzt werden.
// 
// Bausteinbeschreibung:
// Author: Andreas Fast Automation
// Kontakt per LinkedIn: https://www.linkedin.com/in/automation-fast-andreas/
// 
// This project is intended for demonstration purposes and may be used freely.
// 
// Block description:
   VAR_INPUT
      iiStationNo : Int := 1;   // Stationsnummer / Station number
      ixSafetyIsClosed : Bool := true;   // Schutzkreis ist geschlossen / Protective circuit closed
      ixSafetyIsLocked : Bool := true;   // Schutzkreis ist geschlossen und verriegelt / Protective circuit closed and locked
      ixAutoStart : Bool;   // Automatikstart / Automatic start
      ixAutoStop : Bool;   // Automatikstopp / Automatic stop
      ixSinglePulse : Bool;   // Einzelschritt (Halbautomatik) / Single step (semi-automatic)
      ixReset : Bool;   // Station rücksetzen/Grundstellungsfahrt starten / Reset station / start homing
      ixAck : Bool;   // Quittieren / Acknowledge
      ixError : Bool;   // Störung vorhanden / Fault present
      ixRobotsStopped : Bool := true;   // Roboter sind angehalten / Robots stopped
   END_VAR
   VAR_IN_OUT
      iqudtMachine : "typeMachine";
      iqudtStation : "typeStation";
      iqudtSetup : "typeManualMoveSetup";
      iqudtPlcErrMsg : "typePlcErrMsg";
      iqudtHmiErrMsg : "typeHmiErrMsg";
   END_VAR
   VAR
      sxTrigReset : Bool;
      sxTrigSinglePulse : Bool;
      sxTrigHomingDone : Bool;
      sxTrigAutomaticMode : Bool;
      sxTrigTap : Bool;
      sxTrigAuto : Bool;
      sinstAlarmHandler : "AlarmHandler";
   END_VAR
   VAR_TEMP
      txHomingDone : Bool;
      txSqInError : Bool;
      txSqAllInHome : Bool;
      txSqAllJogDone : Bool;
      txSqsAreWaiting : Bool;
      txSinglePulse : Bool;
      txResetReleaseCycle : Bool;   // Rücksetze ReleaseCycle, wenn mindestens eine Schrittkette eine Störung hat und alle anderen den Halteschritt erreicht haben / Reset ReleaseCycle when at least one sequence has a fault and all other sequences have reached the stop step
      txDefinedStopByMachineError : Bool;   // Definierter Stop in der Grundstellung, wenn die Maschine eine Störung hat / Controlled stop in the home position when the machine has a fault
   END_VAR
   VAR_TEMP   // added for the SCL form of the ladder/FBD networks
      _w1 : Bool;
      _w2 : Bool;
      _w3 : Bool;
   END_VAR
BEGIN

REGION Network 1: Station ist vorhanden / nicht reserviert / Station present / not reserved
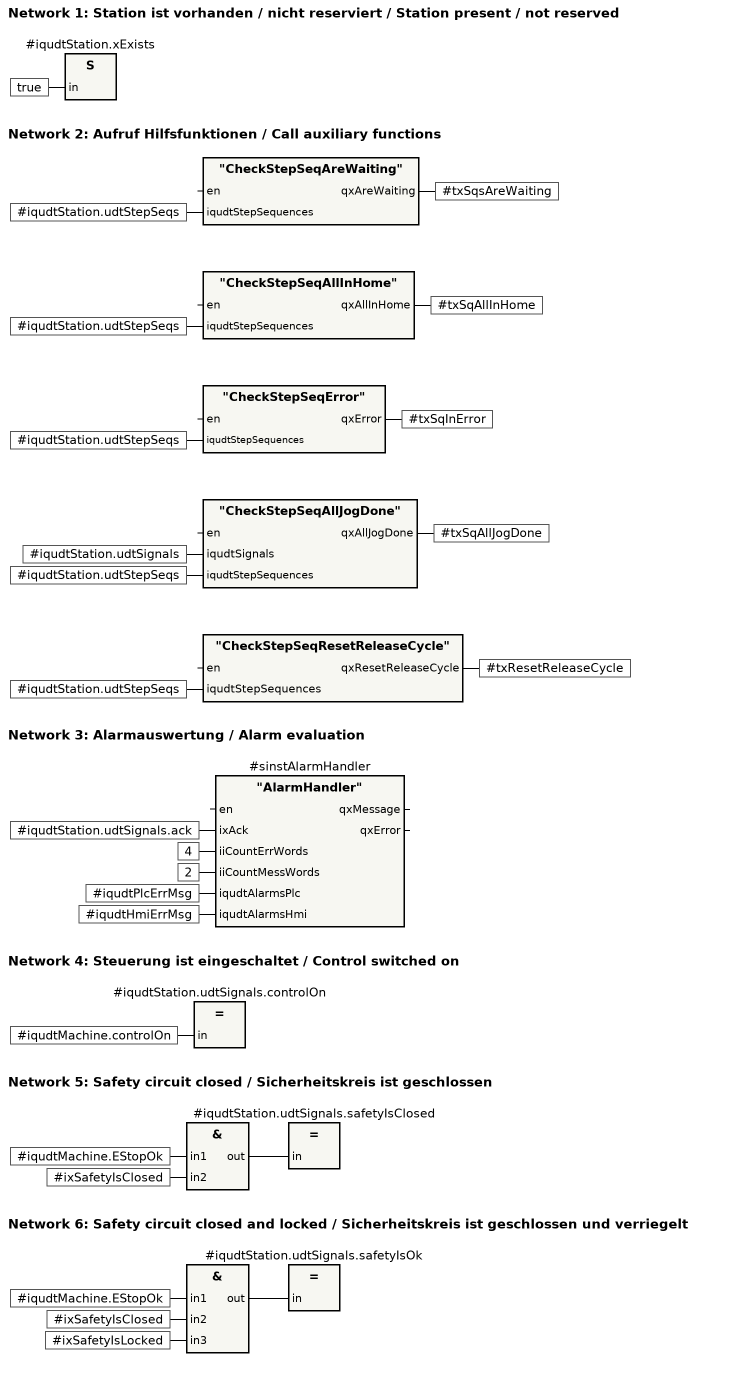
   IF true THEN #iqudtStation.xExists := TRUE; END_IF;
END_REGION

REGION Network 2: Aufruf Hilfsfunktionen / Call auxiliary functions
   "CheckStepSeqAreWaiting"(iqudtStepSequences := #iqudtStation.udtStepSeqs, qxAreWaiting => #txSqsAreWaiting);
   "CheckStepSeqAllInHome"(iqudtStepSequences := #iqudtStation.udtStepSeqs, qxAllInHome => #txSqAllInHome);
   "CheckStepSeqError"(iqudtStepSequences := #iqudtStation.udtStepSeqs, qxError => #txSqInError);
   "CheckStepSeqAllJogDone"(iqudtSignals := #iqudtStation.udtSignals,
                           iqudtStepSequences := #iqudtStation.udtStepSeqs,
                           qxAllJogDone => #txSqAllJogDone);
   "CheckStepSeqResetReleaseCycle"(iqudtStepSequences := #iqudtStation.udtStepSeqs,
                           qxResetReleaseCycle => #txResetReleaseCycle);
END_REGION

REGION Network 3: Alarmauswertung / Alarm evaluation
   #sinstAlarmHandler(ixAck := #iqudtStation.udtSignals.ack,   // "AlarmHandler"
                      iiCountErrWords := 4,
                      iiCountMessWords := 2,
                      iqudtAlarmsPlc := #iqudtPlcErrMsg,
                      iqudtAlarmsHmi := #iqudtHmiErrMsg);
END_REGION

REGION Network 4: Steuerung ist eingeschaltet / Control switched on
   #iqudtStation.udtSignals.controlOn := #iqudtMachine.controlOn;
END_REGION

REGION Network 5: Safety circuit closed / Sicherheitskreis ist geschlossen
   #iqudtStation.udtSignals.safetyIsClosed := #iqudtMachine.EStopOk AND #ixSafetyIsClosed;
END_REGION

REGION Network 6: Safety circuit closed and locked / Sicherheitskreis ist geschlossen und verriegelt
   #iqudtStation.udtSignals.safetyIsOk := #iqudtMachine.EStopOk AND #ixSafetyIsClosed AND #ixSafetyIsLocked;
END_REGION

REGION Network 7: Grundstellungsfahrt auslösen / Initiate homing
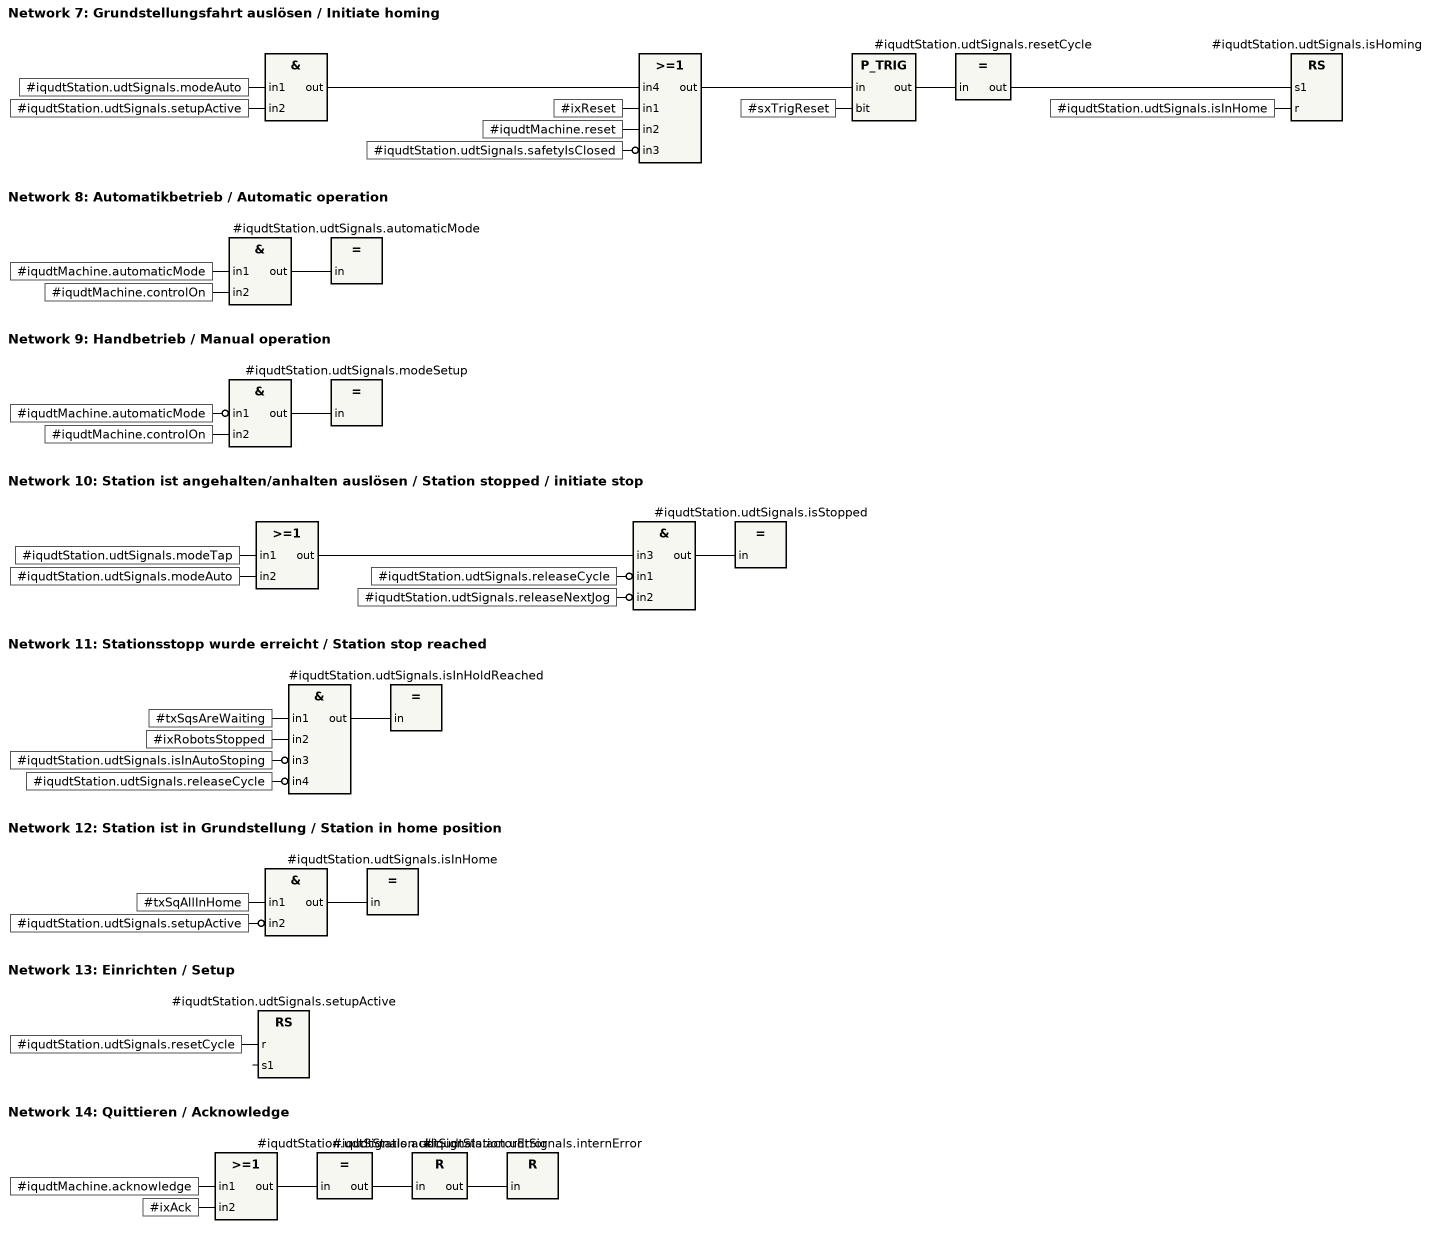
   #_w1 := (#iqudtStation.udtSignals.modeAuto AND #iqudtStation.udtSignals.setupActive) OR #ixReset OR #iqudtMachine.reset OR NOT #iqudtStation.udtSignals.safetyIsClosed;
   #_w2 := #_w1 AND NOT #sxTrigReset;   // rising edge
   #sxTrigReset := #_w1;
   #iqudtStation.udtSignals.resetCycle := #_w2;
   IF #iqudtStation.udtSignals.isInHome THEN
       #iqudtStation.udtSignals.isHoming := FALSE;   // RS flip-flop
   END_IF;
   IF #_w2 THEN #iqudtStation.udtSignals.isHoming := TRUE; END_IF;
END_REGION

REGION Network 8: Automatikbetrieb / Automatic operation
   #iqudtStation.udtSignals.automaticMode := #iqudtMachine.automaticMode AND #iqudtMachine.controlOn;
END_REGION

REGION Network 9: Handbetrieb / Manual operation
   #iqudtStation.udtSignals.modeSetup := NOT #iqudtMachine.automaticMode AND #iqudtMachine.controlOn;
END_REGION

REGION Network 10: Station ist angehalten/anhalten auslösen / Station stopped / initiate stop
   #iqudtStation.udtSignals.isStopped := (#iqudtStation.udtSignals.modeTap OR #iqudtStation.udtSignals.modeAuto) AND NOT #iqudtStation.udtSignals.releaseCycle AND NOT #iqudtStation.udtSignals.releaseNextJog;
END_REGION

REGION Network 11: Stationsstopp wurde erreicht / Station stop reached
   #iqudtStation.udtSignals.isInHoldReached := #txSqsAreWaiting AND #ixRobotsStopped AND NOT #iqudtStation.udtSignals.isInAutoStoping AND NOT #iqudtStation.udtSignals.releaseCycle;
END_REGION

REGION Network 12: Station ist in Grundstellung / Station in home position
   #iqudtStation.udtSignals.isInHome := #txSqAllInHome AND NOT #iqudtStation.udtSignals.setupActive;
END_REGION

REGION Network 13: Einrichten / Setup
   IF #iqudtStation.udtSignals.resetCycle THEN
       #iqudtStation.udtSignals.setupActive := FALSE;   // RS flip-flop
   END_IF;
END_REGION

REGION Network 14: Quittieren / Acknowledge
   #iqudtStation.udtSignals.ack := #iqudtMachine.acknowledge OR #ixAck;
   IF #iqudtStation.udtSignals.ack THEN
       #iqudtStation.udtSignals.actorError := FALSE;
       #iqudtStation.udtSignals.internError := FALSE;
   END_IF;
END_REGION

REGION Network 15: Störung vorhanden / Fault present
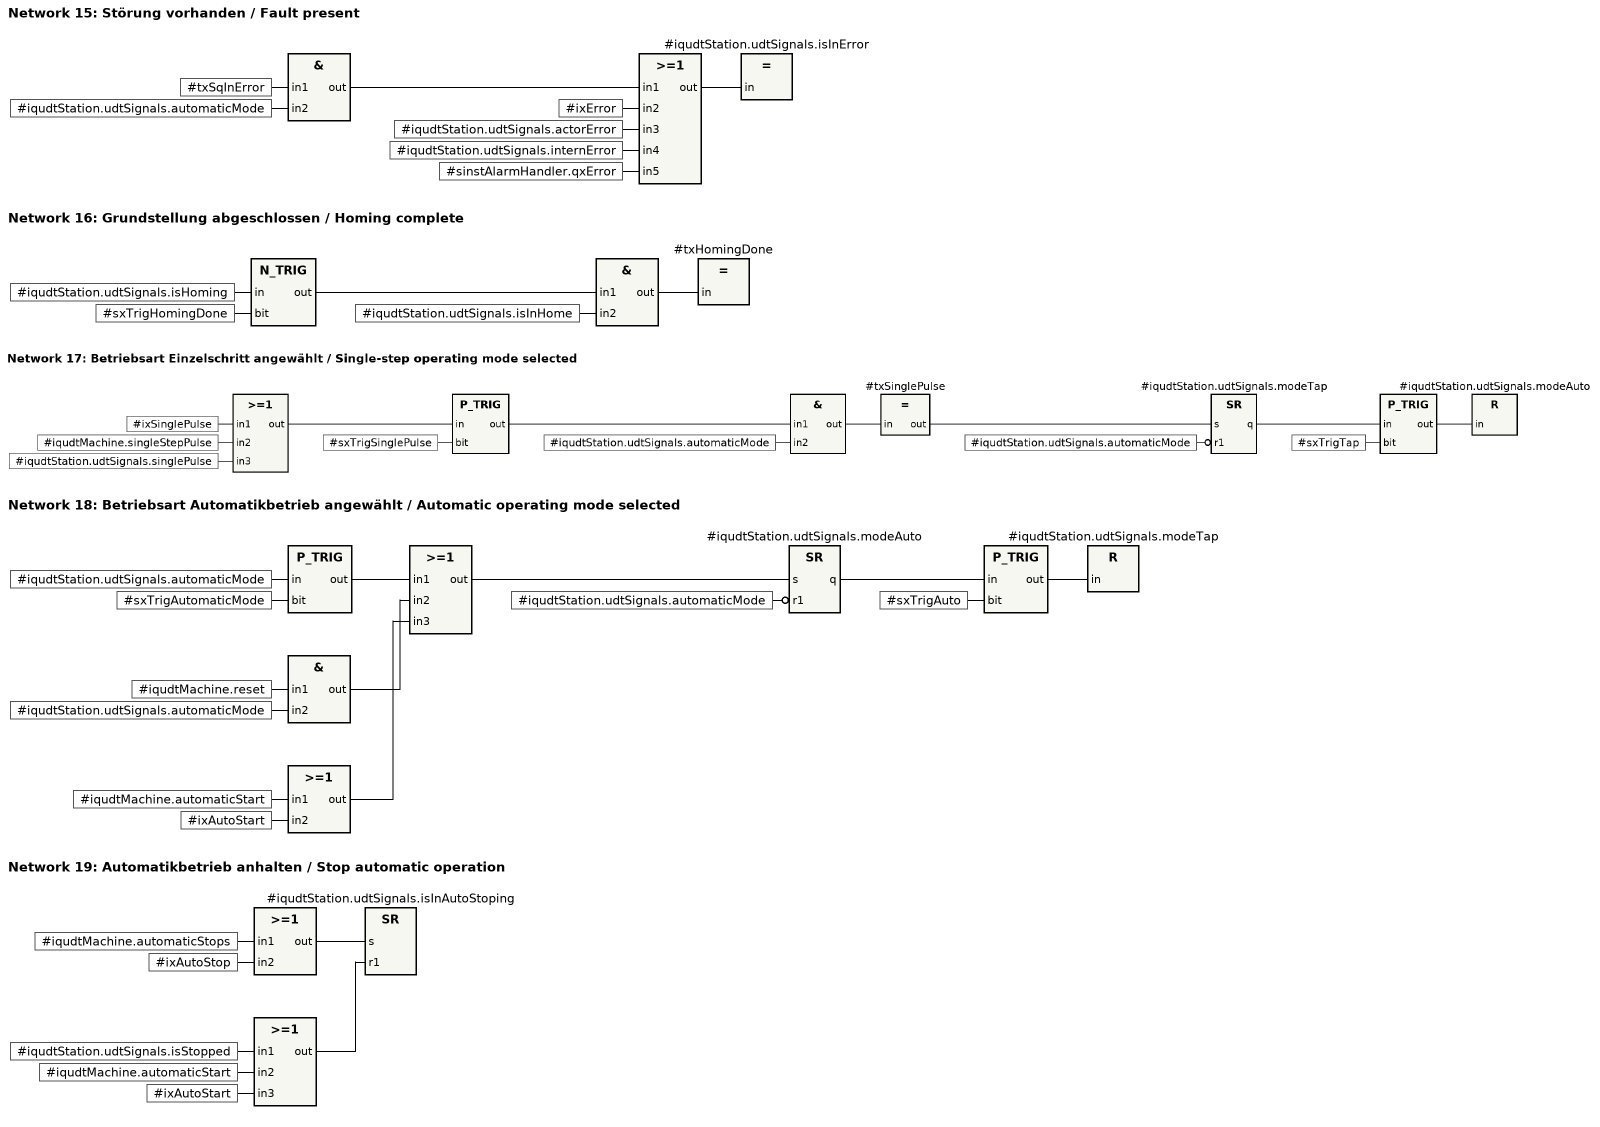
   #iqudtStation.udtSignals.isInError := (#txSqInError AND #iqudtStation.udtSignals.automaticMode) OR #ixError OR #iqudtStation.udtSignals.actorError OR #iqudtStation.udtSignals.internError OR #sinstAlarmHandler.qxError;
END_REGION

REGION Network 16: Grundstellung abgeschlossen / Homing complete
   #_w1 := NOT #iqudtStation.udtSignals.isHoming AND #sxTrigHomingDone;   // falling edge
   #sxTrigHomingDone := #iqudtStation.udtSignals.isHoming;
   #txHomingDone := #_w1 AND #iqudtStation.udtSignals.isInHome;
END_REGION

REGION Network 17: Betriebsart Einzelschritt angewählt / Single-step operating mode selected
   #_w1 := #ixSinglePulse OR #iqudtMachine.singleStepPulse OR #iqudtStation.udtSignals.singlePulse;
   #_w2 := #_w1 AND NOT #sxTrigSinglePulse;   // rising edge
   #sxTrigSinglePulse := #_w1;
   #txSinglePulse := #_w2 AND #iqudtStation.udtSignals.automaticMode;
   IF #txSinglePulse THEN
       #iqudtStation.udtSignals.modeTap := TRUE;   // SR flip-flop
   END_IF;
   IF NOT #iqudtStation.udtSignals.automaticMode THEN #iqudtStation.udtSignals.modeTap := FALSE; END_IF;
   #_w3 := #iqudtStation.udtSignals.modeTap AND NOT #sxTrigTap;   // rising edge
   #sxTrigTap := #iqudtStation.udtSignals.modeTap;
   IF #_w3 THEN #iqudtStation.udtSignals.modeAuto := FALSE; END_IF;
END_REGION

REGION Network 18: Betriebsart Automatikbetrieb angewählt / Automatic operating mode selected
   #_w1 := #iqudtStation.udtSignals.automaticMode AND NOT #sxTrigAutomaticMode;   // rising edge
   #sxTrigAutomaticMode := #iqudtStation.udtSignals.automaticMode;
   IF #_w1 OR (#iqudtMachine.reset AND #iqudtStation.udtSignals.automaticMode) OR #iqudtMachine.automaticStart OR #ixAutoStart THEN
       #iqudtStation.udtSignals.modeAuto := TRUE;   // SR flip-flop
   END_IF;
   IF NOT #iqudtStation.udtSignals.automaticMode THEN #iqudtStation.udtSignals.modeAuto := FALSE; END_IF;
   #_w2 := #iqudtStation.udtSignals.modeAuto AND NOT #sxTrigAuto;   // rising edge
   #sxTrigAuto := #iqudtStation.udtSignals.modeAuto;
   IF #_w2 THEN #iqudtStation.udtSignals.modeTap := FALSE; END_IF;
END_REGION

REGION Network 19: Automatikbetrieb anhalten / Stop automatic operation
   IF #iqudtMachine.automaticStops OR #ixAutoStop THEN
       #iqudtStation.udtSignals.isInAutoStoping := TRUE;   // SR flip-flop
   END_IF;
   IF #iqudtStation.udtSignals.isStopped OR #iqudtMachine.automaticStart OR #ixAutoStart THEN
       #iqudtStation.udtSignals.isInAutoStoping := FALSE;
   END_IF;
END_REGION

REGION Network 20: Halbautomatische Weiterschaltung / Semi-automatic step advance
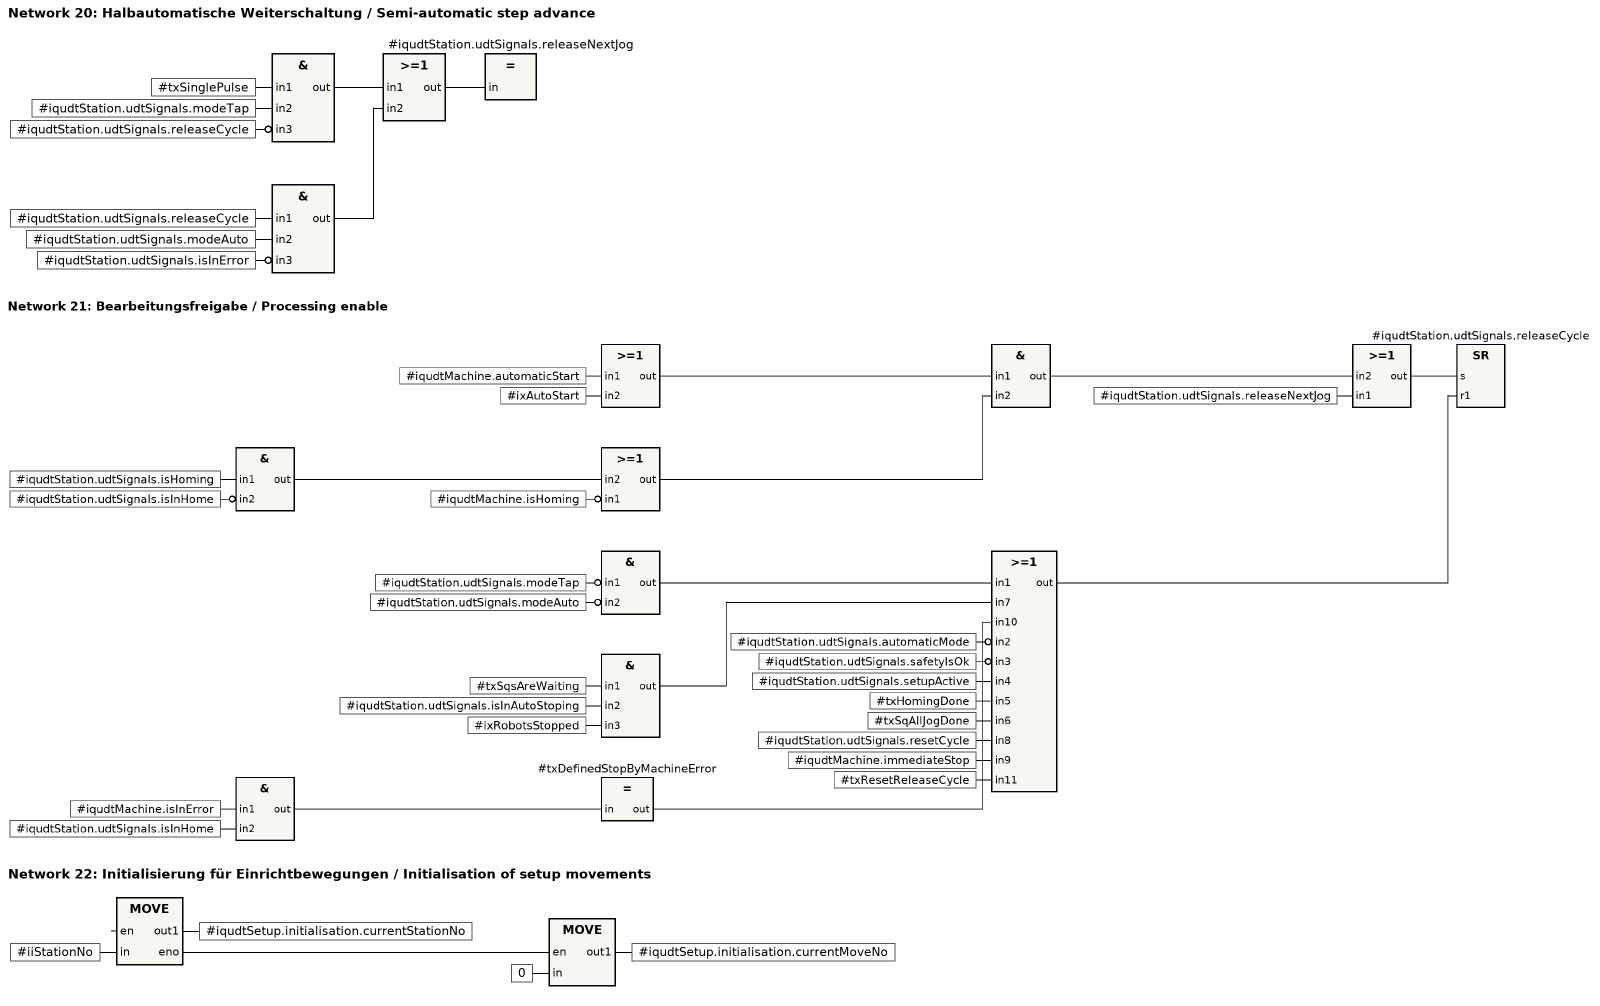
   #iqudtStation.udtSignals.releaseNextJog := (#txSinglePulse AND #iqudtStation.udtSignals.modeTap AND NOT #iqudtStation.udtSignals.releaseCycle) OR (#iqudtStation.udtSignals.releaseCycle AND #iqudtStation.udtSignals.modeAuto AND NOT #iqudtStation.udtSignals.isInError);
END_REGION

REGION Network 21: Bearbeitungsfreigabe / Processing enable
   #txDefinedStopByMachineError := #iqudtMachine.isInError AND #iqudtStation.udtSignals.isInHome;
   IF ((#iqudtMachine.automaticStart OR #ixAutoStart) AND ((#iqudtStation.udtSignals.isHoming AND NOT #iqudtStation.udtSignals.isInHome) OR NOT #iqudtMachine.isHoming)) OR #iqudtStation.udtSignals.releaseNextJog THEN
       #iqudtStation.udtSignals.releaseCycle := TRUE;   // SR flip-flop
   END_IF;
   IF (NOT #iqudtStation.udtSignals.modeTap AND NOT #iqudtStation.udtSignals.modeAuto) OR (#txSqsAreWaiting AND #iqudtStation.udtSignals.isInAutoStoping AND #ixRobotsStopped) OR #txDefinedStopByMachineError OR NOT #iqudtStation.udtSignals.automaticMode OR NOT #iqudtStation.udtSignals.safetyIsOk OR #iqudtStation.udtSignals.setupActive OR #txHomingDone OR #txSqAllJogDone OR #iqudtStation.udtSignals.resetCycle OR #iqudtMachine.immediateStop OR #txResetReleaseCycle THEN
       #iqudtStation.udtSignals.releaseCycle := FALSE;
   END_IF;
END_REGION

REGION Network 22: Initialisierung für Einrichtbewegungen / Initialisation of setup movements
   #iqudtSetup.initialisation.currentStationNo := #iiStationNo;
   #iqudtSetup.initialisation.currentMoveNo := 0;
END_REGION
END_FUNCTION_BLOCK

FUNCTION "CheckStepSeqError" : Void   // FC911, SCL
{ S7_Optimized_Access := 'TRUE' }
VERSION : 0.1
   VAR_OUTPUT
      qxError : Bool;
   END_VAR
   VAR_IN_OUT
      iqudtStepSequences : "typeStepSequences";
   END_VAR
   VAR_TEMP
      tusiCounter : USInt;
   END_VAR
BEGIN
   // Ersteller: Andreas Fast Automation
   // Kontakt per LinkedIn: https://www.linkedin.com/in/automation-fast-andreas/
   //
   // Projekt dient zu Demonstrationszwecken und frei genutzt werden.
   //
   // Bausteinbeschreibung:
   // 

   #qxError := false;



   FOR #tusiCounter := 1 TO "SYS_SQ_MAXSEQUENCES" DO
       // Check for error in stations
       IF #iqudtStepSequences.stepSeq[#tusiCounter].error AND #iqudtStepSequences.stepSeq[#tusiCounter].exists THEN
           #qxError := true;
           RETURN;
       END_IF;
   END_FOR;
END_FUNCTION

FUNCTION "CheckStepSeqAllInHome" : Void   // FC912, SCL
{ S7_Optimized_Access := 'TRUE' }
VERSION : 0.1
   VAR_OUTPUT
      qxAllInHome : Bool;   // Alle Schrittketten in Grundstellung / All sequences in home position
   END_VAR
   VAR_IN_OUT
      iqudtStepSequences : "typeStepSequences";
   END_VAR
   VAR_TEMP
      tusiCounter : USInt;
   END_VAR
BEGIN
   // Ersteller: Andreas Fast Automation
   // Kontakt per LinkedIn: https://www.linkedin.com/in/automation-fast-andreas/
   //
   // Projekt dient zu Demonstrationszwecken und frei genutzt werden.
   //
   // Bausteinbeschreibung:
   // 

   #qxAllInHome := true;



   FOR #tusiCounter := 1 TO "SYS_SQ_MAXSEQUENCES" DO
       // Check for error in stations
       IF NOT #iqudtStepSequences.stepSeq[#tusiCounter].inHome AND #iqudtStepSequences.stepSeq[#tusiCounter].exists THEN
           #qxAllInHome := false;
           RETURN;
       END_IF;
   END_FOR;
END_FUNCTION

FUNCTION "CheckStepSeqAreWaiting" : Void   // FC913, SCL
{ S7_Optimized_Access := 'TRUE' }
VERSION : 0.1
   VAR_OUTPUT
      qxAreWaiting : Bool;   // Warten oder Störung vorhanden / Waiting or in fault state
   END_VAR
   VAR_IN_OUT
      iqudtStepSequences : "typeStepSequences";
   END_VAR
   VAR_TEMP
      tusiCounter : USInt;
   END_VAR
BEGIN
   // Ersteller: Andreas Fast Automation
   // Kontakt per LinkedIn: https://www.linkedin.com/in/automation-fast-andreas/
   //
   // Projekt dient zu Demonstrationszwecken und frei genutzt werden.
   //
   // Bausteinbeschreibung:
   // 

   #qxAreWaiting := true;


   FOR #tusiCounter := 1 TO "SYS_SQ_MAXSEQUENCES" DO
       // Check for error in stations
       IF NOT #iqudtStepSequences.stepSeq[#tusiCounter].isWaiting AND NOT #iqudtStepSequences.stepSeq[#tusiCounter].error AND #iqudtStepSequences.stepSeq[#tusiCounter].exists THEN
           #qxAreWaiting := false;
           RETURN;
       END_IF;
   END_FOR;
END_FUNCTION

FUNCTION "CheckStepSeqAllJogDone" : Void   // FC914, SCL
{ S7_Optimized_Access := 'TRUE' }
VERSION : 0.1
   VAR_OUTPUT
      qxAllJogDone : Bool;   // Alle Schrittketten haben halbautomatische Weiterschaltung abgeschlossen / All sequences have completed semi-automatic step advance
   END_VAR
   VAR_IN_OUT
      iqudtSignals : "typeStationSignals";
      iqudtStepSequences : "typeStepSequences";
   END_VAR
   VAR_TEMP
      tusiCounter : USInt;
   END_VAR
BEGIN
   // Ersteller: Andreas Fast Automation
   // Kontakt per LinkedIn: https://www.linkedin.com/in/automation-fast-andreas/
   //
   // Projekt dient zu Demonstrationszwecken und frei genutzt werden.
   //
   // Bausteinbeschreibung:
   // 

   #qxAllJogDone := false;

   IF (#iqudtSignals.modeTap AND NOT #iqudtSignals.releaseNextJog) THEN // OR (#signals.modeAuto AND #signals.autoIsStoping) THEN

       #qxAllJogDone := #iqudtSignals.releaseCycle;

       FOR #tusiCounter := 1 TO "SYS_SQ_MAXSEQUENCES" DO
           // Check if step sequence is done and exists
           IF NOT #iqudtStepSequences.stepSeq[#tusiCounter].jogDone AND NOT #iqudtStepSequences.stepSeq[#tusiCounter].isWaiting AND NOT #iqudtStepSequences.stepSeq[#tusiCounter].error  AND #iqudtStepSequences.stepSeq[#tusiCounter].exists THEN
               #qxAllJogDone := false;
               RETURN;
           END_IF;
       END_FOR;
   ELSE
       #qxAllJogDone := false;
   END_IF;
END_FUNCTION

FUNCTION "CheckStepSeqResetReleaseCycle" : Void   // FC917, SCL
{ S7_Optimized_Access := 'TRUE' }
VERSION : 0.1
   VAR_OUTPUT
      qxResetReleaseCycle : Bool;
   END_VAR
   VAR_IN_OUT
      iqudtStepSequences : "typeStepSequences";
   END_VAR
   VAR_TEMP
      tusiCounter : USInt;
   END_VAR
BEGIN
   // Ersteller: Andreas Fast Automation
   // Kontakt per LinkedIn: https://www.linkedin.com/in/automation-fast-andreas/
   //
   // Projekt dient zu Demonstrationszwecken und frei genutzt werden.
   //
   // Bausteinbeschreibung:
   // Wenn eine Kette eine Störung hat und alle anderen Schrittende (JogDone) erreicht haben,
   // wird ReleaseCycle zurückgesetzt.

   #qxResetReleaseCycle := false;


   FOR #tusiCounter := 1 TO "SYS_SQ_MAXSEQUENCES" DO

       // Check for error in step sequence
       IF #iqudtStepSequences.stepSeq[#tusiCounter].exists AND
           #iqudtStepSequences.stepSeq[#tusiCounter].error 
       THEN
           #qxResetReleaseCycle := true;
       END_IF;

       // Check other step sequences for jogDone and not error
       IF #iqudtStepSequences.stepSeq[#tusiCounter].exists AND
           NOT #iqudtStepSequences.stepSeq[#tusiCounter].error AND 
           NOT #iqudtStepSequences.stepSeq[#tusiCounter].jogDone AND
           NOT #iqudtStepSequences.stepSeq[#tusiCounter].isWaiting
       THEN
           #qxResetReleaseCycle := false;
           RETURN;
       END_IF;
   END_FOR;
END_FUNCTION

// folder: 9. Library/9.1 Framework Functions/03_ManualMovement

FUNCTION_BLOCK "ActorManualMovement"   // FB909, FBD
TITLE = Steuerung Einrichtbewegung eines Aktors / Control of an actuator setup movement
{ S7_Optimized_Access := 'TRUE' }
VERSION : 0.1
// Ersteller: Andreas Fast Automation
// Kontakt per LinkedIn: https://www.linkedin.com/in/automation-fast-andreas/
// 
// Das Projekt dient zu Demonstrationszwecken und kann frei genutzt werden.
// 
// Bausteinbeschreibung:
// Author: Andreas Fast Automation
// Kontakt per LinkedIn: https://www.linkedin.com/in/automation-fast-andreas/
// 
// This project is intended for demonstration purposes and may be used freely.
// 
// Block description:
   VAR_INPUT
      ixShowValue : Bool;
      ixIsExecutableRight : Bool;
      ixIsExecutableLeft : Bool;
      ixShowEndPositionRight : Bool;   // Sichtbarkeit rechte Seite / Right side visibility
      ixShowEndPositionLeft : Bool;   // Sichtbarkeit linke Seite / Left side visibility
   END_VAR
   VAR_OUTPUT
      quiManualMoveNo : UInt;
   END_VAR
   VAR_IN_OUT
      iqxManualWorkPos : Bool;   // Manueller Ansteuerbefehl für Arbeitsstellung / Manual working position command
      iqxManualHomePos : Bool;   // Manueller Ansteuerbefehl für Grundstellung / Manual home position command
      iqudtActor : "typeActor";
      iqudtSignals : "typeStationSignals";
      iqudtManualMovement : "typeManualMovements";
   END_VAR
   VAR
      suiManualMovementNo : UInt;
      susiStationNo : USInt;
      suiMoveNoInStation : UInt;
   END_VAR
   VAR_TEMP
      txInitialised : Bool;
      txRelease : Bool;
   END_VAR
   VAR_TEMP   // added for the SCL form of the ladder/FBD networks
      _w1 : Bool;
   END_VAR
BEGIN

REGION Network 1: Initialisierungsprozess für eine Einrichtfunktion / Initialisation process for a setup function
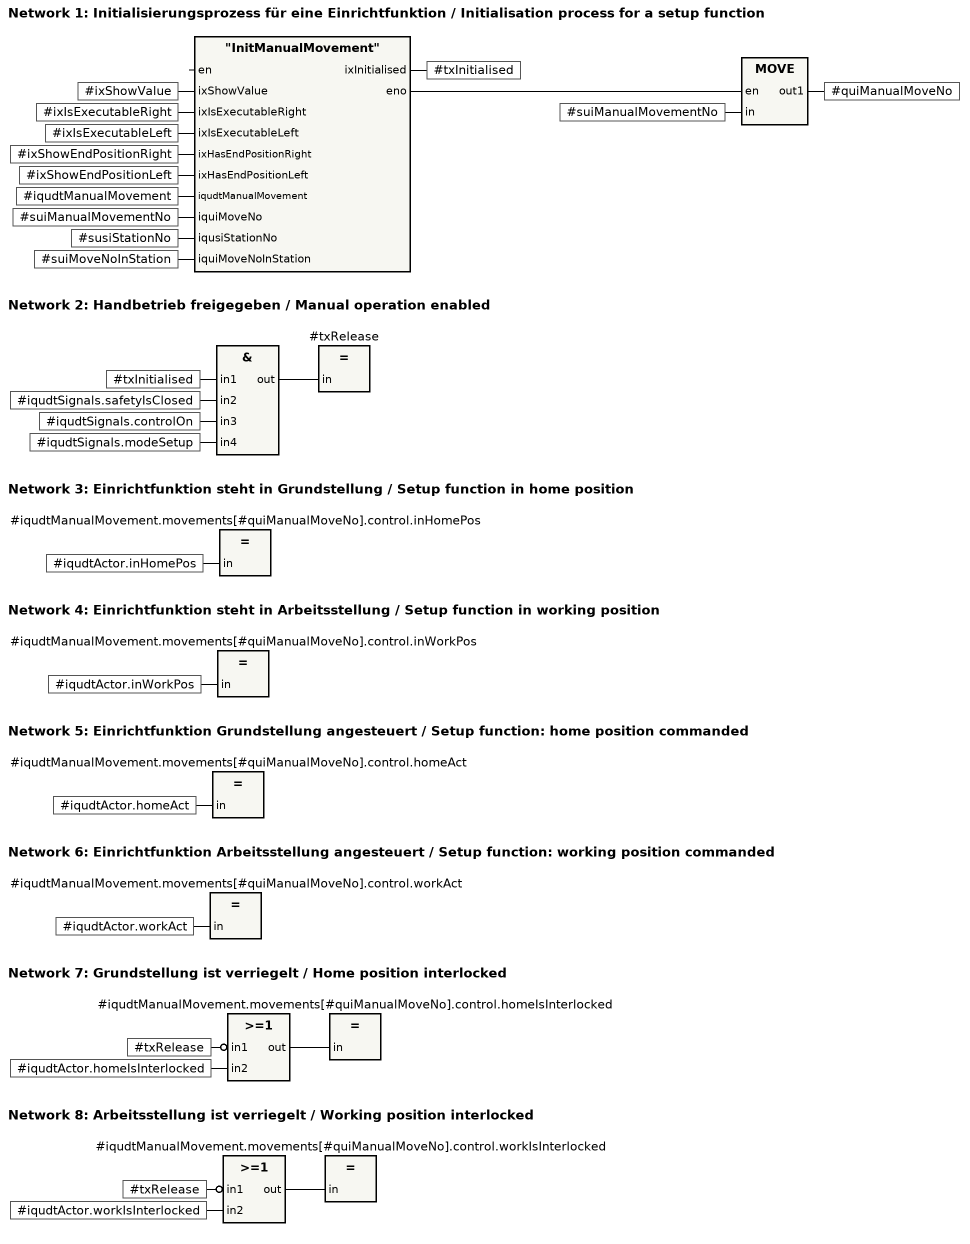
   "InitManualMovement"(ixShowValue := #ixShowValue,
                        ixIsExecutableRight := #ixIsExecutableRight,
                        ixIsExecutableLeft := #ixIsExecutableLeft,
                        ixHasEndPositionRight := #ixShowEndPositionRight,
                        ixHasEndPositionLeft := #ixShowEndPositionLeft,
                        iqudtManualMovement := #iqudtManualMovement,
                        iquiMoveNo := #suiManualMovementNo,
                        iqusiStationNo := #susiStationNo,
                        iquiMoveNoInStation := #suiMoveNoInStation,
                        ixInitialised => #txInitialised,
                        ENO => #_w1);
   IF #_w1 THEN #quiManualMoveNo := #suiManualMovementNo; END_IF;
END_REGION

REGION Network 2: Handbetrieb freigegeben / Manual operation enabled
   #txRelease := #txInitialised AND #iqudtSignals.safetyIsClosed AND #iqudtSignals.controlOn AND #iqudtSignals.modeSetup;
END_REGION

REGION Network 3: Einrichtfunktion steht in Grundstellung / Setup function in home position
   #iqudtManualMovement.movements[#quiManualMoveNo].control.inHomePos := #iqudtActor.inHomePos;
END_REGION

REGION Network 4: Einrichtfunktion steht in Arbeitsstellung / Setup function in working position
   #iqudtManualMovement.movements[#quiManualMoveNo].control.inWorkPos := #iqudtActor.inWorkPos;
END_REGION

REGION Network 5: Einrichtfunktion Grundstellung angesteuert / Setup function: home position commanded
   #iqudtManualMovement.movements[#quiManualMoveNo].control.homeAct := #iqudtActor.homeAct;
END_REGION

REGION Network 6: Einrichtfunktion Arbeitsstellung angesteuert / Setup function: working position commanded
   #iqudtManualMovement.movements[#quiManualMoveNo].control.workAct := #iqudtActor.workAct;
END_REGION

REGION Network 7: Grundstellung ist verriegelt / Home position interlocked
   #iqudtManualMovement.movements[#quiManualMoveNo].control.homeIsInterlocked := NOT #txRelease OR #iqudtActor.homeIsInterlocked;
END_REGION

REGION Network 8: Arbeitsstellung ist verriegelt / Working position interlocked
   #iqudtManualMovement.movements[#quiManualMoveNo].control.workIsInterlocked := NOT #txRelease OR #iqudtActor.workIsInterlocked;
END_REGION

REGION Network 9: Manuelle Bewegungsansteuerung des Aktors zurücksetzen / Reset manual actuator movement command
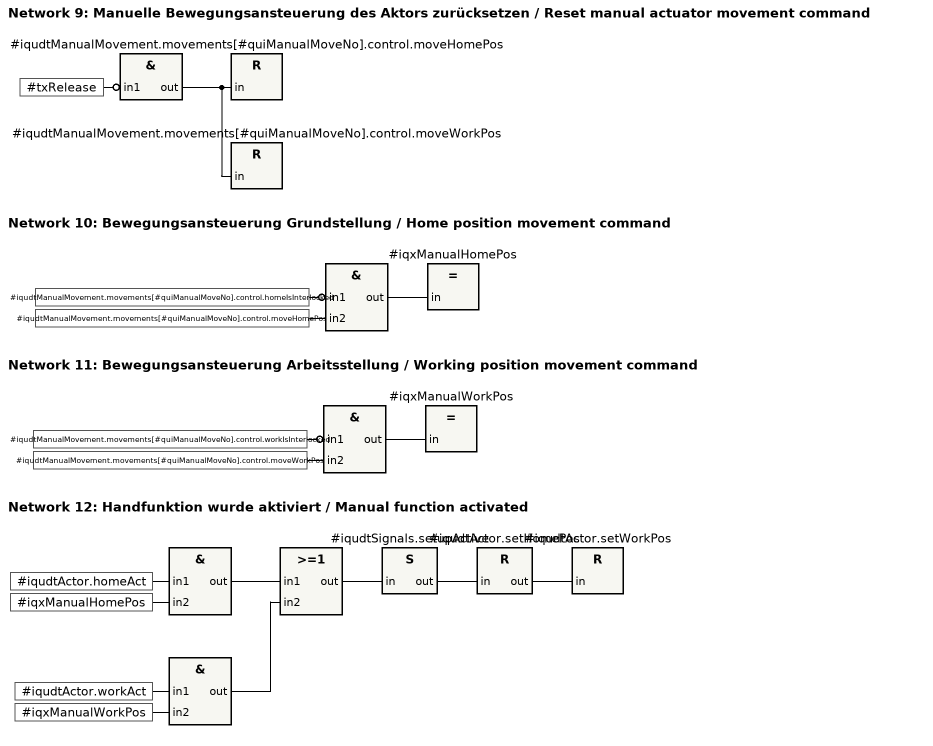
   IF NOT #txRelease THEN
       #iqudtManualMovement.movements[#quiManualMoveNo].control.moveHomePos := FALSE;
       #iqudtManualMovement.movements[#quiManualMoveNo].control.moveWorkPos := FALSE;
   END_IF;
END_REGION

REGION Network 10: Bewegungsansteuerung Grundstellung / Home position movement command
   #iqxManualHomePos := NOT #iqudtManualMovement.movements[#quiManualMoveNo].control.homeIsInterlocked AND #iqudtManualMovement.movements[#quiManualMoveNo].control.moveHomePos;
END_REGION

REGION Network 11: Bewegungsansteuerung Arbeitsstellung / Working position movement command
   #iqxManualWorkPos := NOT #iqudtManualMovement.movements[#quiManualMoveNo].control.workIsInterlocked AND #iqudtManualMovement.movements[#quiManualMoveNo].control.moveWorkPos;
END_REGION

REGION Network 12: Handfunktion wurde aktiviert / Manual function activated
   IF (#iqudtActor.homeAct AND #iqxManualHomePos) OR (#iqudtActor.workAct AND #iqxManualWorkPos) THEN
       #iqudtSignals.setupActive := TRUE;
       #iqudtActor.setHomePos := FALSE;
       #iqudtActor.setWorkPos := FALSE;
   END_IF;
END_REGION
END_FUNCTION_BLOCK

FUNCTION "InitManualMovement" : Void   // FC907, FBD
TITLE = Initialisierungsprozess für eine Einrichtfunktion / Initialisation process for a setup function
{ S7_Optimized_Access := 'TRUE' }
VERSION : 0.1
// Ersteller: Andreas Fast Automation
// Kontakt per LinkedIn: https://www.linkedin.com/in/automation-fast-andreas/
// 
// Das Projekt dient zu Demonstrationszwecken und kann frei genutzt werden.
// 
// Bausteinbeschreibung:
// Author: Andreas Fast Automation
// Kontakt per LinkedIn: https://www.linkedin.com/in/automation-fast-andreas/
// 
// This project is intended for demonstration purposes and may be used freely.
// 
// Block description:
   VAR_INPUT
      ixShowValue : Bool;   // Zeige Dezimalanzeige / Show decimal display
      ixIsExecutableRight : Bool;   // Ist ausführbar rechte Seite / Right side executable
      ixIsExecutableLeft : Bool;   // Ist ausführbar linke Seite / Left side executable
      ixHasEndPositionRight : Bool;   // Zeige Endposition rechte Seite / Display right end position
      ixHasEndPositionLeft : Bool;   // Zeige Endposition linke Seite / Display left end position
   END_VAR
   VAR_OUTPUT
      ixInitialised : Bool;
   END_VAR
   VAR_IN_OUT
      iqudtManualMovement : "typeManualMovements";
      iquiMoveNo : UInt;
      iqusiStationNo : USInt;
      iquiMoveNoInStation : UInt;
   END_VAR
   VAR_TEMP   // added for the SCL form of the ladder/FBD networks
      _w1 : Bool;
   END_VAR
BEGIN

REGION Network 1: Plausibilitätsprüfung/Initialisierung läuft / Plausibility check/initialisation in progress
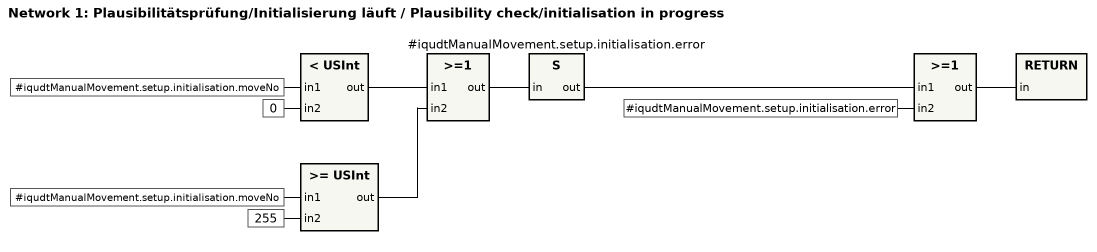
   #_w1 := (#iqudtManualMovement.setup.initialisation.moveNo < 0) OR (#iqudtManualMovement.setup.initialisation.moveNo >= 255);
   IF #_w1 THEN #iqudtManualMovement.setup.initialisation.error := TRUE; END_IF;
   IF #_w1 OR #iqudtManualMovement.setup.initialisation.error THEN
       ENO := TRUE;
       RETURN;
   END_IF;
END_REGION

REGION Network 2: Initialisierung / Initialisation
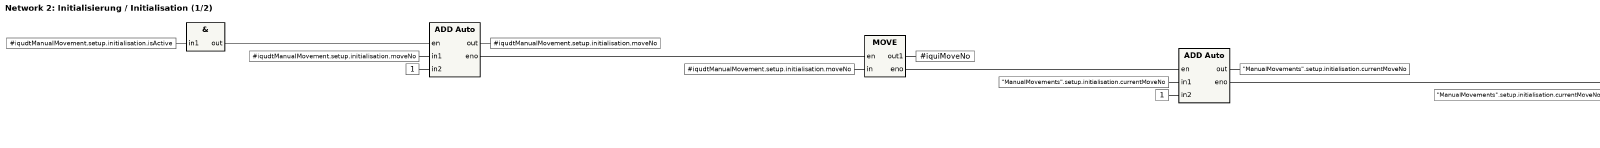
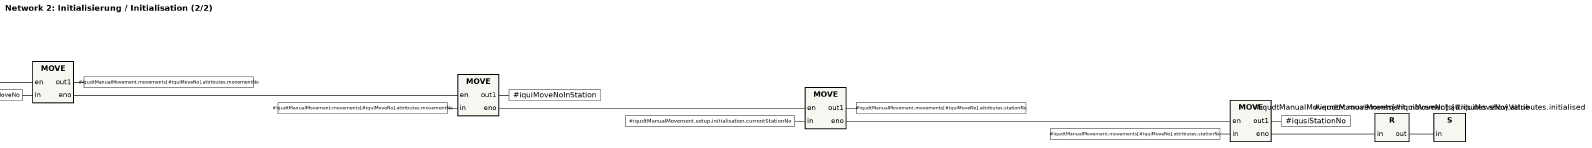
   IF #iqudtManualMovement.setup.initialisation.isActive THEN
       #iqudtManualMovement.setup.initialisation.moveNo := #iqudtManualMovement.setup.initialisation.moveNo + 1;
       #iquiMoveNo := #iqudtManualMovement.setup.initialisation.moveNo;
       "ManualMovements".setup.initialisation.currentMoveNo := "ManualMovements".setup.initialisation.currentMoveNo + 1;
       #iqudtManualMovement.movements[#iquiMoveNo].attributes.movementNo := "ManualMovements".setup.initialisation.currentMoveNo;
       #iquiMoveNoInStation := #iqudtManualMovement.movements[#iquiMoveNo].attributes.movementNo;
       #iqudtManualMovement.movements[#iquiMoveNo].attributes.stationNo := #iqudtManualMovement.setup.initialisation.currentStationNo;
       #iqusiStationNo := #iqudtManualMovement.movements[#iquiMoveNo].attributes.stationNo;
       #iqudtManualMovement.movements[#iquiMoveNo].attributes.showValue := FALSE;
       #iqudtManualMovement.movements[#iquiMoveNo].attributes.initialised := TRUE;
   END_IF;
END_REGION

REGION Network 3: Initialisierung abgeschlossen? / Initialisation complete?
